  01:  // Wait for responce received
       IF ( _responseReceived )
       THEN
         // reset response received flag
        _responseReceived := FALSE;
         // update state flags
         OnUpdateStateFlags(_response.State);
         // update state flags
         OnApplyOutCmd(_response.State);
                
         // Done, Aborted or Error ?
         IF (_response.State >= CmdMessageState.DONE )
         THEN
           // Update the WorAreas in user defined system datas 
           AxesGroup.SystemData.UpdateWorAreas( Caller       := THIS^,
                                                SystemTime   := AxesGroup.State.SystemTime,
                                                WorkAreaNo   := OutCmd.WorkAreaNoReturn, 
                                                WorkAreaData := OutCmd.WorkAreaData);                     
           // set timeout
           SetTimeout(PT := _timeoutCmd, rTimer := _timerCmd);
           // inc step counter
          _stepCmd := _stepCmd + 1; 
         END_IF
       END_IF


  02: IF ( NOT Execute)
      THEN
        Reset();
      END_IF     

ELSE
  // invalid step
  SetError( ErrorID := RobotLibraryErrorIdEnum.ERR_INVALID_STEP, Overwrite := TRUE );
END_CASE


// Reset FB
IF ( NOT Execute )
THEN
  Reset(); 
END_IF
                
END_METHOD

METHOD PROTECTED OnUpdateStateFlags
VAR_INPUT
  /// Command message state
  State : CmdMessageState;
END_VAR
                  // Reset State flags
Done := FALSE;

CASE State OF

  // No operation or process is active
  CmdMessageState.EMPTY               :;
  // Created but not yet started
  CmdMessageState.CREATED             :;
  // Buffered and awaiting execution
  CmdMessageState.BUFFERED            : CommandBuffered    := TRUE;             
  // Buffered in planner for future execution
  CmdMessageState.BUFFERED_IN_PLANNER : CommandBuffered    := TRUE; 
  // Currently active and in progress
  CmdMessageState.ACTIVE              :;                                 
  // Interrupted and awaiting continuation
  CmdMessageState.INTERRUPTED         :;     
  // Requested for abort
  CmdMessageState.ABORT_REQUEST       :;
  // Successfully completed
  CmdMessageState.DONE                : Done               := TRUE;
                                        Busy               := FALSE;
  // Aborted before completion
  CmdMessageState.ABORTED             : Busy               := FALSE;
  // Encountered an error during execution
  CmdMessageState.ERROR               : Error              := TRUE;
                                        Busy               := FALSE;
END_CASE
                
END_METHOD

METHOD INTERNAL ParseResponsePayload : DINT
VAR_INPUT
  /// Response data
  ResponseData : RobotLibraryResponseDataFB;
  /// Timestamp
  Timestamp    : SystemTime;  
END_VAR
VAR
  /// Parameter count
 _parameterCnt : DINT;
END_VAR
// Table 6-200: Received CMD payload (RC to PLC) of "ReadWorkArea"
// --------------------------
// Header
// --------------------------
// Byte 00 : USINT   - ParSeq | State     
// Byte 01 : SINT    - AlarmMessageSeverity    
// Byte 02 : UINT    - AlarmMessageCode HB
// Byte 03 :         - AlarmMessageCode LB
// --------------------------
// Datablock
// --------------------------
// Byte 04 : USINT    - WorkAreaNo;
// Byte 05 : BYTE     - Reserved;
// Byte 06 : DATE     - Data.Date HW HB;
// Byte 07 :          - Data.Date HW LB;
// Byte 08 : IED_TIME - Data.Time HW HB;
// Byte 09 :          - Data.Time HW LB;
// Byte 10 :          - Data.Time LW HB;
// Byte 11 :          - Data.Time LW LB;
// Byte 12 : USINT    - Data.AreaType;
// Byte 13 : BOOL     - Data.AreaMode;
// Byte 14 : USINT    - Data.ReactionMode;
// Byte 15 : BOOL     - Data.ActiveModification;
// Byte 16 : USINT    - Data.DefinitionMode;
// Byte 17 : USINT    - Data.FrameNo;
// Byte 18 : REAL     - Data.ZeroPointX HW HB;
// Byte 19 :          - Data.ZeroPointX HW LB;
// Byte 20 :          - Data.ZeroPointX LW HB;
// Byte 21 :          - Data.ZeroPointX LW LB;
// Byte 22 : REAL     - Data.ZeroPointY HW HB;
// Byte 23 :          - Data.ZeroPointY HW LB;
// Byte 24 :          - Data.ZeroPointY LW HB;
// Byte 25 :          - Data.ZeroPointY LW LB;
// Byte 26 : REAL     - Data.ZeroPointZ HW HB;
// Byte 27 :          - Data.ZeroPointZ HW LB;
// Byte 28 :          - Data.ZeroPointZ LW HB;
// Byte 29 :          - Data.ZeroPointZ LW LB;
// Byte 30 : REAL     - Data.X1 HW HB;
// Byte 31 :          - Data.X1 HW LB;
// Byte 32 :          - Data.X1 LW HB;
// Byte 33 :          - Data.X1 LW LB;
// Byte 34 : REAL     - Data.X2 HW HB;
// Byte 35 :          - Data.X2 HW LB;
// Byte 36 :          - Data.X2 LW HB;
// Byte 37 :          - Data.X2 LW LB;
// Byte 38 : REAL     - Data.Y1 HW HB;
// Byte 39 :          - Data.Y1 HW LB;
// Byte 40 :          - Data.Y1 LW HB;
// Byte 41 :          - Data.Y1 LW LB;
// Byte 42 : REAL     - Data.Y2 HW HB;
// Byte 43 :          - Data.Y2 HW LB;
// Byte 44 :          - Data.Y2 LW HB;
// Byte 45 :          - Data.Y2 LW LB;
// Byte 46 : REAL     - Data.Z1 HW HB;
// Byte 47 :          - Data.Z1 HW LB;
// Byte 48 :          - Data.Z1 LW HB;
// Byte 49 :          - Data.Z1 LW LB;
// Byte 50 : REAL     - Data.Z2 HW HB;
// Byte 51 :          - Data.Z2 HW LB;
// Byte 52 :          - Data.Z2 LW HB;
// Byte 53 :          - Data.Z2 LW LB;
// Byte 54 : REAL     - Data.Radius HW HB;
// Byte 55 :          - Data.Radius HW LB;
// Byte 56 :          - Data.Radius LW HB;
// Byte 57 :          - Data.Radius LW LB;
// Byte 58 : REAL     - Data.JointLowerLimit.J1 HW HB;
// Byte 59 :          - Data.JointLowerLimit.J1 HW LB;
// Byte 60 :          - Data.JointLowerLimit.J1 LW HB;
// Byte 61 :          - Data.JointLowerLimit.J1 LW LB;
// Byte 62 : REAL     - Data.JointLowerLimit.J2 HW HB;
// Byte 63 :          - Data.JointLowerLimit.J2 HW LB;
// Byte 64 :          - Data.JointLowerLimit.J2 LW HB;
// Byte 65 :          - Data.JointLowerLimit.J2 LW LB;
// Byte 66 : REAL     - Data.JointLowerLimit.J3 HW HB;
// Byte 67 :          - Data.JointLowerLimit.J3 HW LB;
// Byte 68 :          - Data.JointLowerLimit.J3 LW HB;
// Byte 69 :          - Data.JointLowerLimit.J3 LW LB;
// Byte 70 : REAL     - Data.JointLowerLimit.J4 HW HB;
// Byte 71 :          - Data.JointLowerLimit.J4 HW LB;
// Byte 72 :          - Data.JointLowerLimit.J4 LW HB;
// Byte 73 :          - Data.JointLowerLimit.J4 LW LB;
// Byte 74 : REAL     - Data.JointLowerLimit.J5 HW HB;
// Byte 75 :          - Data.JointLowerLimit.J5 HW LB;
// Byte 76 :          - Data.JointLowerLimit.J5 LW HB;
// Byte 77 :          - Data.JointLowerLimit.J5 LW LB;
// Byte 78 : REAL     - Data.JointLowerLimit.J6 HW HB;
// Byte 79 :          - Data.JointLowerLimit.J6 HW LB;
// Byte 80 :          - Data.JointLowerLimit.J6 LW HB;
// Byte 81 :          - Data.JointLowerLimit.J6 LW LB;
// Byte 82 : REAL     - Data.JointLowerLimit.E1 HW HB;
// Byte 83 :          - Data.JointLowerLimit.E1 HW LB;
// Byte 84 :          - Data.JointLowerLimit.E1 LW HB;
// Byte 85 :          - Data.JointLowerLimit.E1 LW LB;
// Byte 86 : REAL     - Data.JointUpperLimit.J1 HW HB;
// Byte 87 :          - Data.JointUpperLimit.J1 HW LB;
// Byte 88 :          - Data.JointUpperLimit.J1 LW HB;
// Byte 89 :          - Data.JointUpperLimit.J1 LW LB;
// Byte 90 : REAL     - Data.JointUpperLimit.J2 HW HB;
// Byte 91 :          - Data.JointUpperLimit.J2 HW LB;
// Byte 92 :          - Data.JointUpperLimit.J2 LW HB;
// Byte 93 :          - Data.JointUpperLimit.J2 LW LB;
// Byte 94 : REAL     - Data.JointUpperLimit.J3 HW HB;
// Byte 95 :          - Data.JointUpperLimit.J3 HW LB;
// Byte 96 :          - Data.JointUpperLimit.J3 LW HB;
// Byte 97 :          - Data.JointUpperLimit.J3 LW LB;
// Byte 98 : REAL     - Data.JointUpperLimit.J4 HW HB;
// Byte 99 :          - Data.JointUpperLimit.J4 HW LB;
// Byte 100:          - Data.JointUpperLimit.J4 LW HB;
// Byte 101:          - Data.JointUpperLimit.J4 LW LB;
// Byte 102: REAL     - Data.JointUpperLimit.J5 HW HB;
// Byte 103:          - Data.JointUpperLimit.J5 HW LB;
// Byte 104:          - Data.JointUpperLimit.J5 LW HB;
// Byte 105:          - Data.JointUpperLimit.J5 LW LB;
// Byte 106: REAL     - Data.JointUpperLimit.J6 HW HB;
// Byte 107:          - Data.JointUpperLimit.J6 HW LB;
// Byte 108:          - Data.JointUpperLimit.J6 LW HB;
// Byte 109:          - Data.JointUpperLimit.J6 LW LB;
// Byte 110: REAL     - Data.JointUpperLimit.E1 HW HB;
// Byte 111:          - Data.JointUpperLimit.E1 HW LB;
// Byte 112:          - Data.JointUpperLimit.E1 LW HB;
// Byte 113:          - Data.JointUpperLimit.E1 LW LB;
// Byte 114: REAL     - Data.JointLowerLimit.E2 HW HB;
// Byte 115:          - Data.JointLowerLimit.E2 HW LB;
// Byte 116:          - Data.JointLowerLimit.E2 LW HB;
// Byte 117:          - Data.JointLowerLimit.E2 LW LB;
// Byte 118: REAL     - Data.JointLowerLimit.E3 HW HB;
// Byte 119:          - Data.JointLowerLimit.E3 HW LB;
// Byte 120:          - Data.JointLowerLimit.E3 LW HB;
// Byte 121:          - Data.JointLowerLimit.E3 LW LB;
// Byte 122: REAL     - Data.JointLowerLimit.E4 HW HB;
// Byte 123:          - Data.JointLowerLimit.E4 HW LB;
// Byte 124:          - Data.JointLowerLimit.E4 LW HB;
// Byte 125:          - Data.JointLowerLimit.E4 LW LB;
// Byte 126: REAL     - Data.JointLowerLimit.E5 HW HB;
// Byte 127:          - Data.JointLowerLimit.E5 HW LB;
// Byte 128:          - Data.JointLowerLimit.E5 LW HB;
// Byte 129:          - Data.JointLowerLimit.E5 LW LB;
// Byte 130: REAL     - Data.JointLowerLimit.E6 HW HB;
// Byte 131:          - Data.JointLowerLimit.E6 HW LB;
// Byte 132:          - Data.JointLowerLimit.E6 LW HB;
// Byte 133:          - Data.JointLowerLimit.E6 LW LB;
// Byte 134: REAL     - Data.JointUpperLimit.E2 HW HB;
// Byte 135:          - Data.JointUpperLimit.E2 HW LB;
// Byte 136:          - Data.JointUpperLimit.E2 LW HB;
// Byte 137:          - Data.JointUpperLimit.E2 LW LB;
// Byte 138: REAL     - Data.JointUpperLimit.E3 HW HB;
// Byte 139:          - Data.JointUpperLimit.E3 HW LB;
// --------------------------
                  // call base implementation to parse the header from payload buffer
ResponseData.PayloadPtr := SUPER^.ParseResponsePayload(ResponseData := ResponseData, Timestamp := Timestamp);

// copy parsed header to response
_response.ParSeq               := _rspHeader.ParSeq;
_response.State                := _rspHeader.State;
_response.AlarmMessageSeverity := _rspHeader.AlarmMessageSeverity;
_response.AlarmMessageCode     := _rspHeader.AlarmMessageCode;


// Check payload remaining ? 
IF ( ResponseData.IsPayloadRemaining)
THEN  
  // Get Response.WorkAreaNoReturn
 _response.WorkAreaNoReturn := ResponseData.GetUsint();
  // inc parameter counter
 _parameterCnt := _parameterCnt + 1;
END_IF


// Check payload remaining ? 
IF ( ResponseData.IsPayloadRemaining)
THEN  
  // Get Response.Reserve
 _response.Reserve := ResponseData.GetByte();
  // inc parameter counter
 _parameterCnt := _parameterCnt + 1;
END_IF


// Check payload remaining ? 
IF ( ResponseData.IsPayloadRemaining)
THEN  
  // Get Response.WorkAreaData.Timestamp.IEC_DATE
 _response.WorkAreaData.Timestamp.IEC_DATE := ResponseData.GetIecDate();
  // inc parameter counter
 _parameterCnt := _parameterCnt + 1;
END_IF


// Check payload remaining ? 
IF ( ResponseData.IsPayloadRemaining)
THEN  
  // Get Response.WorkAreaData.Timestamp.IEC_TIME
 _response.WorkAreaData.Timestamp.IEC_TIME := ResponseData.GetIecTime();
  // inc parameter counter
 _parameterCnt := _parameterCnt + 1;
END_IF


// Check payload remaining ? 
IF ( ResponseData.IsPayloadRemaining)
THEN  
  // Get Response.WorkAreaData.AreaType
 _response.WorkAreaData.AreaType := ResponseData.GetUsint();
  // inc parameter counter
 _parameterCnt := _parameterCnt + 1;
END_IF


// Check payload remaining ? 
IF ( ResponseData.IsPayloadRemaining)
THEN  
  // Get Response.WorkAreaData.AreaMode
 _response.WorkAreaData.AreaMode := ResponseData.GetBool();
  // inc parameter counter
 _parameterCnt := _parameterCnt + 1;
END_IF


// Check payload remaining ? 
IF ( ResponseData.IsPayloadRemaining)
THEN  
  // Get Response.WorkAreaData.ReactionMode
 _response.WorkAreaData.ReactionMode := ResponseData.GetUsint();
  // inc parameter counter
 _parameterCnt := _parameterCnt + 1;
END_IF


// Check payload remaining ? 
IF ( ResponseData.IsPayloadRemaining)
THEN  
  // Get Response.WorkAreaData.ActiveModification
 _response.WorkAreaData.ActiveModification := ResponseData.GetBool();
  // inc parameter counter
 _parameterCnt := _parameterCnt + 1;
END_IF


// Check payload remaining ? 
IF ( ResponseData.IsPayloadRemaining)
THEN  
  // Get Response.WorkAreaData.DefinitionMode
 _response.WorkAreaData.DefinitionMode := ResponseData.GetUsint();
  // inc parameter counter
 _parameterCnt := _parameterCnt + 1;
END_IF


// Check payload remaining ? 
IF ( ResponseData.IsPayloadRemaining)
THEN  
  // Get Response.WorkAreaData.FrameNo
 _response.WorkAreaData.FrameNo := ResponseData.GetUsint();
  // inc parameter counter
 _parameterCnt := _parameterCnt + 1;
END_IF


// Check payload remaining ? 
IF ( ResponseData.IsPayloadRemaining)
THEN  
  // Get Response.WorkAreaData.ZeroPointX
 _response.WorkAreaData.ZeroPointX := ResponseData.GetReal();
  // inc parameter counter
 _parameterCnt := _parameterCnt + 1;
END_IF


// Check payload remaining ? 
IF ( ResponseData.IsPayloadRemaining)
THEN  
  // Get Response.WorkAreaData.ZeroPointY
 _response.WorkAreaData.ZeroPointY := ResponseData.GetReal();
  // inc parameter counter
 _parameterCnt := _parameterCnt + 1;
END_IF


// Check payload remaining ? 
IF ( ResponseData.IsPayloadRemaining)
THEN  
  // Get Response.WorkAreaData.ZeroPointZ
 _response.WorkAreaData.ZeroPointZ := ResponseData.GetReal();
  // inc parameter counter
 _parameterCnt := _parameterCnt + 1;
END_IF


// Check payload remaining ? 
IF ( ResponseData.IsPayloadRemaining)
THEN  
  // Get Response.WorkAreaData.X.LowerLimit
 _response.WorkAreaData.X.LowerLimit := ResponseData.GetReal();
  // inc parameter counter
 _parameterCnt := _parameterCnt + 1;
END_IF


// Check payload remaining ? 
IF ( ResponseData.IsPayloadRemaining)
THEN  
  // Get Response.WorkAreaData.X.UpperLimit
 _response.WorkAreaData.X.UpperLimit := ResponseData.GetReal();
  // inc parameter counter
 _parameterCnt := _parameterCnt + 1;
END_IF


// Check payload remaining ? 
IF ( ResponseData.IsPayloadRemaining)
THEN  
  // Get Response.WorkAreaData.Y.LowerLimit
 _response.WorkAreaData.Y.LowerLimit := ResponseData.GetReal();
  // inc parameter counter
 _parameterCnt := _parameterCnt + 1;
END_IF


// Check payload remaining ? 
IF ( ResponseData.IsPayloadRemaining)
THEN  
  // Get Response.WorkAreaData.Y.UpperLimit
 _response.WorkAreaData.Y.UpperLimit := ResponseData.GetReal();
  // inc parameter counter
 _parameterCnt := _parameterCnt + 1;
END_IF


// Check payload remaining ? 
IF ( ResponseData.IsPayloadRemaining)
THEN  
  // Get Response.WorkAreaData.Z.LowerLimit
 _response.WorkAreaData.Z.LowerLimit := ResponseData.GetReal();
  // inc parameter counter
 _parameterCnt := _parameterCnt + 1;
END_IF


// Check payload remaining ? 
IF ( ResponseData.IsPayloadRemaining)
THEN  
  // Get Response.WorkAreaData.Z.UpperLimit
 _response.WorkAreaData.Z.UpperLimit := ResponseData.GetReal();
  // inc parameter counter
 _parameterCnt := _parameterCnt + 1;
END_IF


// Check payload remaining ? 
IF ( ResponseData.IsPayloadRemaining)
THEN  
  // Get Response.WorkAreaData.Radiust
 _response.WorkAreaData.Radius := ResponseData.GetReal();
  // inc parameter counter
 _parameterCnt := _parameterCnt + 1;
END_IF


// Check payload remaining ? 
IF ( ResponseData.IsPayloadRemaining)
THEN  
  // Get Response.WorkAreaData.J1Limit.LowerLimit
 _response.WorkAreaData.J1Limit.LowerLimit := ResponseData.GetReal();
  // inc parameter counter
 _parameterCnt := _parameterCnt + 1;
END_IF


// Check payload remaining ? 
IF ( ResponseData.IsPayloadRemaining)
THEN  
  // Get Response.WorkAreaData.J2Limit.LowerLimit
 _response.WorkAreaData.J2Limit.LowerLimit := ResponseData.GetReal();
  // inc parameter counter
 _parameterCnt := _parameterCnt + 1;
END_IF


// Check payload remaining ? 
IF ( ResponseData.IsPayloadRemaining)
THEN  
  // Get Response.WorkAreaData.J3Limit.LowerLimit
 _response.WorkAreaData.J3Limit.LowerLimit := ResponseData.GetReal();
  // inc parameter counter
 _parameterCnt := _parameterCnt + 1;
END_IF


// Check payload remaining ? 
IF ( ResponseData.IsPayloadRemaining)
THEN  
  // Get Response.WorkAreaData.J4Limit.LowerLimit
 _response.WorkAreaData.J4Limit.LowerLimit := ResponseData.GetReal();
  // inc parameter counter
 _parameterCnt := _parameterCnt + 1;
END_IF


// Check payload remaining ? 
IF ( ResponseData.IsPayloadRemaining)
THEN  
  // Get Response.WorkAreaData.J5Limit.LowerLimit
 _response.WorkAreaData.J5Limit.LowerLimit := ResponseData.GetReal();
  // inc parameter counter
 _parameterCnt := _parameterCnt + 1;
END_IF


// Check payload remaining ? 
IF ( ResponseData.IsPayloadRemaining)
THEN  
  // Get Response.WorkAreaData.J6Limit.LowerLimit
 _response.WorkAreaData.J6Limit.LowerLimit := ResponseData.GetReal();
  // inc parameter counter
 _parameterCnt := _parameterCnt + 1;
END_IF


// Check payload remaining ? 
IF ( ResponseData.IsPayloadRemaining)
THEN  
  // Get Response.WorkAreaData.E1Limit.LowerLimit
 _response.WorkAreaData.E1Limit.LowerLimit := ResponseData.GetReal();
  // inc parameter counter
 _parameterCnt := _parameterCnt + 1;
END_IF


// Check payload remaining ? 
IF ( ResponseData.IsPayloadRemaining)
THEN  
  // Get Response.WorkAreaData.J1Limit.UpperLimit
 _response.WorkAreaData.J1Limit.UpperLimit := ResponseData.GetReal();
  // inc parameter counter
 _parameterCnt := _parameterCnt + 1;
END_IF


// Check payload remaining ? 
IF ( ResponseData.IsPayloadRemaining)
THEN  
  // Get Response.WorkAreaData.J2Limit.UpperLimit
 _response.WorkAreaData.J2Limit.UpperLimit := ResponseData.GetReal();
  // inc parameter counter
 _parameterCnt := _parameterCnt + 1;
END_IF


// Check payload remaining ? 
IF ( ResponseData.IsPayloadRemaining)
THEN  
  // Get Response.WorkAreaData.J3Limit.UpperLimit
 _response.WorkAreaData.J3Limit.UpperLimit := ResponseData.GetReal();
  // inc parameter counter
 _parameterCnt := _parameterCnt + 1;
END_IF


// Check payload remaining ? 
IF ( ResponseData.IsPayloadRemaining)
THEN  
  // Get Response.WorkAreaData.J4Limit.UpperLimit
 _response.WorkAreaData.J4Limit.UpperLimit := ResponseData.GetReal();
  // inc parameter counter
 _parameterCnt := _parameterCnt + 1;
END_IF


// Check payload remaining ? 
IF ( ResponseData.IsPayloadRemaining)
THEN  
  // Get Response.WorkAreaData.J5Limit.UpperLimit
 _response.WorkAreaData.J5Limit.UpperLimit := ResponseData.GetReal();
  // inc parameter counter
 _parameterCnt := _parameterCnt + 1;
END_IF


// Check payload remaining ? 
IF ( ResponseData.IsPayloadRemaining)
THEN  
  // Get Response.WorkAreaData.J6Limit.UpperLimit
 _response.WorkAreaData.J6Limit.UpperLimit := ResponseData.GetReal();
  // inc parameter counter
 _parameterCnt := _parameterCnt + 1;
END_IF


// Check payload remaining ? 
IF ( ResponseData.IsPayloadRemaining)
THEN  
  // Get Response.WorkAreaData.E1Limit.UpperLimit
 _response.WorkAreaData.E1Limit.UpperLimit := ResponseData.GetReal();
  // inc parameter counter
 _parameterCnt := _parameterCnt + 1;
END_IF


// Check payload remaining ? 
IF ( ResponseData.IsPayloadRemaining)
THEN  
  // Get Response.WorkAreaData.E2Limit.LowerLimit
 _response.WorkAreaData.E2Limit.LowerLimit := ResponseData.GetReal();
  // inc parameter counter
 _parameterCnt := _parameterCnt + 1;
END_IF


// Check payload remaining ? 
IF ( ResponseData.IsPayloadRemaining)
THEN  
  // Get Response.WorkAreaData.E3Limit.LowerLimit
 _response.WorkAreaData.E3Limit.LowerLimit := ResponseData.GetReal();
  // inc parameter counter
 _parameterCnt := _parameterCnt + 1;
END_IF


// Check payload remaining ? 
IF ( ResponseData.IsPayloadRemaining)
THEN  
  // Get Response.WorkAreaData.E4Limit.LowerLimit
 _response.WorkAreaData.E4Limit.LowerLimit := ResponseData.GetReal();
  // inc parameter counter
 _parameterCnt := _parameterCnt + 1;
END_IF


// Check payload remaining ? 
IF ( ResponseData.IsPayloadRemaining)
THEN  
  // Get Response.WorkAreaData.E5Limit.LowerLimit
 _response.WorkAreaData.E5Limit.LowerLimit := ResponseData.GetReal();
  // inc parameter counter
 _parameterCnt := _parameterCnt + 1;
END_IF


// Check payload remaining ? 
IF ( ResponseData.IsPayloadRemaining)
THEN  
  // Get Response.WorkAreaData.E6Limit.LowerLimit
 _response.WorkAreaData.E6Limit.LowerLimit := ResponseData.GetReal();
  // inc parameter counter
 _parameterCnt := _parameterCnt + 1;
END_IF


// Check payload remaining ? 
IF ( ResponseData.IsPayloadRemaining)
THEN  
  // Get Response.WorkAreaData.E2Limit.UpperLimit
 _response.WorkAreaData.E2Limit.UpperLimit := ResponseData.GetReal();
  // inc parameter counter
 _parameterCnt := _parameterCnt + 1;
END_IF


// Check payload remaining ? 
IF ( ResponseData.IsPayloadRemaining)
THEN  
  // Get Response.WorkAreaData.E3Limit.UpperLimit
 _response.WorkAreaData.E3Limit.UpperLimit := ResponseData.GetReal();
  // inc parameter counter
 _parameterCnt := _parameterCnt + 1;
END_IF


// Check payload remaining ? 
IF ( ResponseData.IsPayloadRemaining)
THEN  
  // Get Response.WorkAreaData.E4Limit.UpperLimit
 _response.WorkAreaData.E4Limit.UpperLimit := ResponseData.GetReal();
  // inc parameter counter
 _parameterCnt := _parameterCnt + 1;
END_IF


// Check payload remaining ? 
IF ( ResponseData.IsPayloadRemaining)
THEN  
  // Get Response.WorkAreaData.E5Limit.UpperLimit
 _response.WorkAreaData.E5Limit.UpperLimit := ResponseData.GetReal();
  // inc parameter counter
 _parameterCnt := _parameterCnt + 1;
END_IF


// Check payload remaining ? 
IF ( ResponseData.IsPayloadRemaining)
THEN  
  // Get Response.WorkAreaData.E6Limit.UpperLimit
 _response.WorkAreaData.E6Limit.UpperLimit := ResponseData.GetReal();
  // inc parameter counter
 _parameterCnt := _parameterCnt + 1;
END_IF


// Check payload remaining ? 
IF ( ResponseData.IsPayloadRemaining)
THEN  
  // Get Response.DataChanged
 _response.DataChanged := ResponseData.GetBool();
  // inc parameter counter
 _parameterCnt := _parameterCnt + 1;
END_IF



// Create logging
ParseResponsePayloadLog(ResponseData := ResponseData, Timestamp := Timestamp, ParameterCnt := _parameterCnt);
                
END_METHOD

METHOD INTERNAL ParseResponsePayloadLog
VAR_INPUT
  /// Response data
  ResponseData : RobotLibraryResponseDataFB;
  /// Timestamp
  Timestamp    : SystemTime;  
  /// Parameter count
  ParameterCnt : DINT;
END_VAR
                  // Create log entry for Parameter start
CreateLogMessagePara1 ( Timestamp   := Timestamp,
                        MessageType := MessageType.CMD,
                        Severity    := Severity.DEBUG,
                        MessageCode := 0,
                        MessageText := '{1} parameter(s) to parse from the response data:',
                        Para1       := DINT_TO_STRING(ParameterCnt));
                        

// Return if no parameter is remaining...
IF ( ParameterCnt = 0 ) THEN RETURN; END_IF
// dec remaining parameter(s)                        
ParameterCnt := ParameterCnt - 1;
// Create log entry for WorkAreaNoReturn
CreateLogMessagePara1 ( Timestamp   := Timestamp,
                        MessageType := MessageType.CMD,
                        Severity    := Severity.DEBUG,
                        MessageCode := 0,
                        MessageText := 'Response.WorkAreaNoReturn = {1}',
                        Para1       :=  USINT_TO_STRING(_response.WorkAreaNoReturn));


// Return if no parameter is remaining...
IF ( ParameterCnt = 0 ) THEN RETURN; END_IF
// dec remaining parameter(s)                        
ParameterCnt := ParameterCnt - 1;
// Create log entry for Reserve
CreateLogMessagePara1 ( Timestamp   := Timestamp,
                        MessageType := MessageType.CMD,
                        Severity    := Severity.DEBUG,
                        MessageCode := 0,
                        MessageText := 'Response.Reserve = {1}',
                        Para1       :=  BYTE_TO_STRING(_response.Reserve));


// Return if no parameter is remaining...
IF ( ParameterCnt = 0 ) THEN RETURN; END_IF
// dec remaining parameter(s)                        
ParameterCnt := ParameterCnt - 1;
// Create log entry for WorkAreaData.Timestamp.IEC_DATE
CreateLogMessagePara1 ( Timestamp   := Timestamp,
                        MessageType := MessageType.CMD,
                        Severity    := Severity.DEBUG,
                        MessageCode := 0,
                        MessageText := 'Response.WorkAreaData.Timestamp.IEC_DATE = {1}',
                        Para1       :=  IEC_DATE_TO_STRING(_response.WorkAreaData.Timestamp.IEC_DATE));


// Return if no parameter is remaining...
IF ( ParameterCnt = 0 ) THEN RETURN; END_IF
// dec remaining parameter(s)                        
ParameterCnt := ParameterCnt - 1;
// Create log entry for WorkAreaData.Timestamp.IEC_TIME
CreateLogMessagePara1 ( Timestamp   := Timestamp,
                        MessageType := MessageType.CMD,
                        Severity    := Severity.DEBUG,
                        MessageCode := 0,
                        MessageText := 'Response.WorkAreaData.Timestamp.IEC_TIME = {1}',
                        Para1       :=  IEC_TIME_TO_STRING(_response.WorkAreaData.Timestamp.IEC_TIME));


// Return if no parameter is remaining...
IF ( ParameterCnt = 0 ) THEN RETURN; END_IF
// dec remaining parameter(s)                        
ParameterCnt := ParameterCnt - 1;
// Create log entry for WorkAreaData.AreaType
CreateLogMessagePara1 ( Timestamp   := Timestamp,
                        MessageType := MessageType.CMD,
                        Severity    := Severity.DEBUG,
                        MessageCode := 0,
                        MessageText := 'Response.WorkAreaData.AreaType = {1}',
                        Para1       :=  USINT_TO_STRING(_response.WorkAreaData.AreaType));


// Return if no parameter is remaining...
IF ( ParameterCnt = 0 ) THEN RETURN; END_IF
// dec remaining parameter(s)                        
ParameterCnt := ParameterCnt - 1;
// Create log entry for WorkAreaData.AreaMode
CreateLogMessagePara1 ( Timestamp   := Timestamp,
                        MessageType := MessageType.CMD,
                        Severity    := Severity.DEBUG,
                        MessageCode := 0,
                        MessageText := 'Response.WorkAreaData.AreaMode = {1}',
                        Para1       :=  BOOL_TO_STRING(_response.WorkAreaData.AreaMode));
                        

// Return if no parameter is remaining...
IF ( ParameterCnt = 0 ) THEN RETURN; END_IF
// dec remaining parameter(s)                        
ParameterCnt := ParameterCnt - 1;
// Create log entry for WorkAreaData.ReactionMode
CreateLogMessagePara1 ( Timestamp   := Timestamp,
                        MessageType := MessageType.CMD,
                        Severity    := Severity.DEBUG,
                        MessageCode := 0,
                        MessageText := 'Response.WorkAreaData.ReactionMode = {1}',
                        Para1       :=  WORK_AREA_REACTION_MODE_TO_STRING(_response.WorkAreaData.ReactionMode));


// Return if no parameter is remaining...
IF ( ParameterCnt = 0 ) THEN RETURN; END_IF
// dec remaining parameter(s)                        
ParameterCnt := ParameterCnt - 1;
// Create log entry for WorkAreaData.ActiveModification
CreateLogMessagePara1 ( Timestamp   := Timestamp,
                        MessageType := MessageType.CMD,
                        Severity    := Severity.DEBUG,
                        MessageCode := 0,
                        MessageText := 'Response.WorkAreaData.ActiveModification = {1}',
                        Para1       :=  BOOL_TO_STRING(_response.WorkAreaData.ActiveModification));


// Return if no parameter is remaining...
IF ( ParameterCnt = 0 ) THEN RETURN; END_IF
// dec remaining parameter(s)                        
ParameterCnt := ParameterCnt - 1;
// Create log entry for WorkAreaData.DefinitionMode
CreateLogMessagePara1 ( Timestamp   := Timestamp,
                        MessageType := MessageType.CMD,
                        Severity    := Severity.DEBUG,
                        MessageCode := 0,
                        MessageText := 'Response.WorkAreaData.DefinitionMode = {1}',
                        Para1       := DEFINITION_MODE_TO_STRING(_response.WorkAreaData.DefinitionMode));


// Return if no parameter is remaining...
IF ( ParameterCnt = 0 ) THEN RETURN; END_IF
// dec remaining parameter(s)                        
ParameterCnt := ParameterCnt - 1;
// Create log entry for WorkAreaData.FrameNo
CreateLogMessagePara1 ( Timestamp   := Timestamp,
                        MessageType := MessageType.CMD,
                        Severity    := Severity.DEBUG,
                        MessageCode := 0,
                        MessageText := 'Response.WorkAreaData.FrameNo = {1}',
                        Para1       :=  USINT_TO_STRING(_response.WorkAreaData.FrameNo));


// Return if no parameter is remaining...
IF ( ParameterCnt = 0 ) THEN RETURN; END_IF
// dec remaining parameter(s)                        
ParameterCnt := ParameterCnt - 1;
// Create log entry for WorkAreaData.ZeroPointX
CreateLogMessagePara1 ( Timestamp   := Timestamp,
                        MessageType := MessageType.CMD,
                        Severity    := Severity.DEBUG,
                        MessageCode := 0,
                        MessageText := 'Response.WorkAreaData.ZeroPointX = {1}',
                        Para1       :=  REAL_TO_STRING(_response.WorkAreaData.ZeroPointX));


// Return if no parameter is remaining...
IF ( ParameterCnt = 0 ) THEN RETURN; END_IF
// dec remaining parameter(s)                        
ParameterCnt := ParameterCnt - 1;
// Create log entry for WorkAreaData.ZeroPointY
CreateLogMessagePara1 ( Timestamp   := Timestamp,
                        MessageType := MessageType.CMD,
                        Severity    := Severity.DEBUG,
                        MessageCode := 0,
                        MessageText := 'Response.WorkAreaData.ZeroPointY = {1}',
                        Para1       :=  REAL_TO_STRING(_response.WorkAreaData.ZeroPointY));


// Return if no parameter is remaining...
IF ( ParameterCnt = 0 ) THEN RETURN; END_IF
// dec remaining parameter(s)                        
ParameterCnt := ParameterCnt - 1;
// Create log entry for WorkAreaData.ZeroPointZ
CreateLogMessagePara1 ( Timestamp   := Timestamp,
                        MessageType := MessageType.CMD,
                        Severity    := Severity.DEBUG,
                        MessageCode := 0,
                        MessageText := 'Response.WorkAreaData.ZeroPointZ = {1}',
                        Para1       :=  REAL_TO_STRING(_response.WorkAreaData.ZeroPointZ));


// Return if no parameter is remaining...
IF ( ParameterCnt = 0 ) THEN RETURN; END_IF
// dec remaining parameter(s)                        
ParameterCnt := ParameterCnt - 1;
// Create log entry for WorkAreaData.X.LowerLimit
CreateLogMessagePara1 ( Timestamp   := Timestamp,
                        MessageType := MessageType.CMD,
                        Severity    := Severity.DEBUG,
                        MessageCode := 0,
                        MessageText := 'Response.WorkAreaData.X.LowerLimit = {1}',
                        Para1       :=  REAL_TO_STRING(_response.WorkAreaData.X.LowerLimit));


// Return if no parameter is remaining...
IF ( ParameterCnt = 0 ) THEN RETURN; END_IF
// dec remaining parameter(s)                        
ParameterCnt := ParameterCnt - 1;
// Create log entry for WorkAreaData.X.UpperLimit
CreateLogMessagePara1 ( Timestamp   := Timestamp,
                        MessageType := MessageType.CMD,
                        Severity    := Severity.DEBUG,
                        MessageCode := 0,
                        MessageText := 'Response.WorkAreaData.X.UpperLimit = {1}',
                        Para1       :=  REAL_TO_STRING(_response.WorkAreaData.X.UpperLimit));


// Return if no parameter is remaining...
IF ( ParameterCnt = 0 ) THEN RETURN; END_IF
// dec remaining parameter(s)                        
ParameterCnt := ParameterCnt - 1;
// Create log entry for WorkAreaData.Y.LowerLimit
CreateLogMessagePara1 ( Timestamp   := Timestamp,
                        MessageType := MessageType.CMD,
                        Severity    := Severity.DEBUG,
                        MessageCode := 0,
                        MessageText := 'Response.WorkAreaData.Y.LowerLimit = {1}',
                        Para1       :=  REAL_TO_STRING(_response.WorkAreaData.Y.LowerLimit));


// Return if no parameter is remaining...
IF ( ParameterCnt = 0 ) THEN RETURN; END_IF
// dec remaining parameter(s)                        
ParameterCnt := ParameterCnt - 1;
// Create log entry for WorkAreaData.Y.UpperLimit
CreateLogMessagePara1 ( Timestamp   := Timestamp,
                        MessageType := MessageType.CMD,
                        Severity    := Severity.DEBUG,
                        MessageCode := 0,
                        MessageText := 'Response.WorkAreaData.Y.UpperLimit = {1}',
                        Para1       :=  REAL_TO_STRING(_response.WorkAreaData.Y.UpperLimit));


// Return if no parameter is remaining...
IF ( ParameterCnt = 0 ) THEN RETURN; END_IF
// dec remaining parameter(s)                        
ParameterCnt := ParameterCnt - 1;
// Create log entry for WorkAreaData.Z.LowerLimit
CreateLogMessagePara1 ( Timestamp   := Timestamp,
                        MessageType := MessageType.CMD,
                        Severity    := Severity.DEBUG,
                        MessageCode := 0,
                        MessageText := 'Response.WorkAreaData.Z.LowerLimit = {1}',
                        Para1       :=  REAL_TO_STRING(_response.WorkAreaData.Z.LowerLimit));


// Return if no parameter is remaining...
IF ( ParameterCnt = 0 ) THEN RETURN; END_IF
// dec remaining parameter(s)                        
ParameterCnt := ParameterCnt - 1;
// Create log entry for WorkAreaData.Z.UpperLimit
CreateLogMessagePara1 ( Timestamp   := Timestamp,
                        MessageType := MessageType.CMD,
                        Severity    := Severity.DEBUG,
                        MessageCode := 0,
                        MessageText := 'Response.WorkAreaData.Z.UpperLimit = {1}',
                        Para1       :=  REAL_TO_STRING(_response.WorkAreaData.Z.UpperLimit));


// Return if no parameter is remaining...
IF ( ParameterCnt = 0 ) THEN RETURN; END_IF
// dec remaining parameter(s)                        
ParameterCnt := ParameterCnt - 1;
// Create log entry for WorkAreaData.Radius
CreateLogMessagePara1 ( Timestamp   := Timestamp,
                        MessageType := MessageType.CMD,
                        Severity    := Severity.DEBUG,
                        MessageCode := 0,
                        MessageText := 'Response.WorkAreaData.Radius = {1}',
                        Para1       :=  REAL_TO_STRING(_response.WorkAreaData.Radius));


// Return if no parameter is remaining...
IF ( ParameterCnt = 0 ) THEN RETURN; END_IF
// dec remaining parameter(s)                        
ParameterCnt := ParameterCnt - 1;
// Create log entry for WorkAreaData.J1Limit.LowerLimit
CreateLogMessagePara1 ( Timestamp   := Timestamp,
                        MessageType := MessageType.CMD,
                        Severity    := Severity.DEBUG,
                        MessageCode := 0,
                        MessageText := 'Response.WorkAreaData.J1Limit.LowerLimit = {1}',
                        Para1       :=  REAL_TO_STRING(_response.WorkAreaData.J1Limit.LowerLimit));


// Return if no parameter is remaining...
IF ( ParameterCnt = 0 ) THEN RETURN; END_IF
// dec remaining parameter(s)                        
ParameterCnt := ParameterCnt - 1;
// Create log entry for WorkAreaData.J2Limit.LowerLimit
CreateLogMessagePara1 ( Timestamp   := Timestamp,
                        MessageType := MessageType.CMD,
                        Severity    := Severity.DEBUG,
                        MessageCode := 0,
                        MessageText := 'Response.WorkAreaData.J2Limit.LowerLimit = {1}',
                        Para1       :=  REAL_TO_STRING(_response.WorkAreaData.J2Limit.LowerLimit));


// Return if no parameter is remaining...
IF ( ParameterCnt = 0 ) THEN RETURN; END_IF
// dec remaining parameter(s)                        
ParameterCnt := ParameterCnt - 1;
// Create log entry for WorkAreaData.J3Limit.LowerLimit
CreateLogMessagePara1 ( Timestamp   := Timestamp,
                        MessageType := MessageType.CMD,
                        Severity    := Severity.DEBUG,
                        MessageCode := 0,
                        MessageText := 'Response.WorkAreaData.J3Limit.LowerLimit = {1}',
                        Para1       :=  REAL_TO_STRING(_response.WorkAreaData.J3Limit.LowerLimit));

// Return if no parameter is remaining...
IF ( ParameterCnt = 0 ) THEN RETURN; END_IF
// dec remaining parameter(s)                        
ParameterCnt := ParameterCnt - 1;
// Create log entry for WorkAreaData.J4Limit.LowerLimit
CreateLogMessagePara1 ( Timestamp   := Timestamp,
                        MessageType := MessageType.CMD,
                        Severity    := Severity.DEBUG,
                        MessageCode := 0,
                        MessageText := 'Response.WorkAreaData.J4Limit.LowerLimit = {1}',
                        Para1       :=  REAL_TO_STRING(_response.WorkAreaData.J4Limit.LowerLimit));


// Return if no parameter is remaining...
IF ( ParameterCnt = 0 ) THEN RETURN; END_IF
// dec remaining parameter(s)                        
ParameterCnt := ParameterCnt - 1;
// Create log entry for WorkAreaData.J5Limit.LowerLimit
CreateLogMessagePara1 ( Timestamp   := Timestamp,
                        MessageType := MessageType.CMD,
                        Severity    := Severity.DEBUG,
                        MessageCode := 0,
                        MessageText := 'Response.WorkAreaData.J5Limit.LowerLimit = {1}',
                        Para1       :=  REAL_TO_STRING(_response.WorkAreaData.J5Limit.LowerLimit));


// Return if no parameter is remaining...
IF ( ParameterCnt = 0 ) THEN RETURN; END_IF
// dec remaining parameter(s)                        
ParameterCnt := ParameterCnt - 1;
// Create log entry for WorkAreaData.J6Limit.LowerLimit
CreateLogMessagePara1 ( Timestamp   := Timestamp,
                        MessageType := MessageType.CMD,
                        Severity    := Severity.DEBUG,
                        MessageCode := 0,
                        MessageText := 'Response.WorkAreaData.J6Limit.LowerLimit = {1}',
                        Para1       :=  REAL_TO_STRING(_response.WorkAreaData.J6Limit.LowerLimit));


// Return if no parameter is remaining...
IF ( ParameterCnt = 0 ) THEN RETURN; END_IF
// dec remaining parameter(s)                        
ParameterCnt := ParameterCnt - 1;
// Create log entry for WorkAreaData.E1Limit.LowerLimit
CreateLogMessagePara1 ( Timestamp   := Timestamp,
                        MessageType := MessageType.CMD,
                        Severity    := Severity.DEBUG,
                        MessageCode := 0,
                        MessageText := 'Response.WorkAreaData.E1Limit.LowerLimit = {1}',
                        Para1       :=  REAL_TO_STRING(_response.WorkAreaData.E1Limit.LowerLimit));


// Return if no parameter is remaining...
IF ( ParameterCnt = 0 ) THEN RETURN; END_IF
// dec remaining parameter(s)                        
ParameterCnt := ParameterCnt - 1;
// Create log entry for WorkAreaData.J1Limit.UpperLimit
CreateLogMessagePara1 ( Timestamp   := Timestamp,
                        MessageType := MessageType.CMD,
                        Severity    := Severity.DEBUG,
                        MessageCode := 0,
                        MessageText := 'Response.WorkAreaData.J1Limit.UpperLimit = {1}',
                        Para1       :=  REAL_TO_STRING(_response.WorkAreaData.J1Limit.UpperLimit));


// Return if no parameter is remaining...
IF ( ParameterCnt = 0 ) THEN RETURN; END_IF
// dec remaining parameter(s)                        
ParameterCnt := ParameterCnt - 1;
// Create log entry for WorkAreaData.J2Limit.UpperLimit
CreateLogMessagePara1 ( Timestamp   := Timestamp,
                        MessageType := MessageType.CMD,
                        Severity    := Severity.DEBUG,
                        MessageCode := 0,
                        MessageText := 'Response.WorkAreaData.J2Limit.UpperLimit = {1}',
                        Para1       :=  REAL_TO_STRING(_response.WorkAreaData.J2Limit.UpperLimit));


// Return if no parameter is remaining...
IF ( ParameterCnt = 0 ) THEN RETURN; END_IF
// dec remaining parameter(s)                        
ParameterCnt := ParameterCnt - 1;
// Create log entry for WorkAreaData.J3Limit.UpperLimit
CreateLogMessagePara1 ( Timestamp   := Timestamp,
                        MessageType := MessageType.CMD,
                        Severity    := Severity.DEBUG,
                        MessageCode := 0,
                        MessageText := 'Response.WorkAreaData.J3Limit.UpperLimit = {1}',
                        Para1       :=  REAL_TO_STRING(_response.WorkAreaData.J3Limit.UpperLimit));


// Return if no parameter is remaining...
IF ( ParameterCnt = 0 ) THEN RETURN; END_IF
// dec remaining parameter(s)                        
ParameterCnt := ParameterCnt - 1;
// Create log entry for WorkAreaData.J4Limit.UpperLimit
CreateLogMessagePara1 ( Timestamp   := Timestamp,
                        MessageType := MessageType.CMD,
                        Severity    := Severity.DEBUG,
                        MessageCode := 0,
                        MessageText := 'Response.WorkAreaData.J4Limit.UpperLimit = {1}',
                        Para1       :=  REAL_TO_STRING(_response.WorkAreaData.J4Limit.UpperLimit));


// Return if no parameter is remaining...
IF ( ParameterCnt = 0 ) THEN RETURN; END_IF
// dec remaining parameter(s)                        
ParameterCnt := ParameterCnt - 1;
// Create log entry for WorkAreaData.J5Limit.UpperLimit
CreateLogMessagePara1 ( Timestamp   := Timestamp,
                        MessageType := MessageType.CMD,
                        Severity    := Severity.DEBUG,
                        MessageCode := 0,
                        MessageText := 'Response.WorkAreaData.J5Limit.UpperLimit = {1}',
                        Para1       :=  REAL_TO_STRING(_response.WorkAreaData.J5Limit.UpperLimit));


// Return if no parameter is remaining...
IF ( ParameterCnt = 0 ) THEN RETURN; END_IF
// dec remaining parameter(s)                        
ParameterCnt := ParameterCnt - 1;
// Create log entry for WorkAreaData.J6Limit.UpperLimit
CreateLogMessagePara1 ( Timestamp   := Timestamp,
                        MessageType := MessageType.CMD,
                        Severity    := Severity.DEBUG,
                        MessageCode := 0,
                        MessageText := 'Response.WorkAreaData.J6Limit.UpperLimit = {1}',
                        Para1       :=  REAL_TO_STRING(_response.WorkAreaData.J6Limit.UpperLimit));


// Return if no parameter is remaining...
IF ( ParameterCnt = 0 ) THEN RETURN; END_IF
// dec remaining parameter(s)                        
ParameterCnt := ParameterCnt - 1;
// Create log entry for WorkAreaData.E1Limit.UpperLimit
CreateLogMessagePara1 ( Timestamp   := Timestamp,
                        MessageType := MessageType.CMD,
                        Severity    := Severity.DEBUG,
                        MessageCode := 0,
                        MessageText := 'Response.WorkAreaData.E1Limit.UpperLimit = {1}',
                        Para1       :=  REAL_TO_STRING(_response.WorkAreaData.E1Limit.UpperLimit));


// Return if no parameter is remaining...
IF ( ParameterCnt = 0 ) THEN RETURN; END_IF
// dec remaining parameter(s)                        
ParameterCnt := ParameterCnt - 1;
// Create log entry for WorkAreaData.E2Limit.LowerLimit
CreateLogMessagePara1 ( Timestamp   := Timestamp,
                        MessageType := MessageType.CMD,
                        Severity    := Severity.DEBUG,
                        MessageCode := 0,
                        MessageText := 'Response.WorkAreaData.E2Limit.LowerLimit = {1}',
                        Para1       :=  REAL_TO_STRING(_response.WorkAreaData.E2Limit.LowerLimit));


// Return if no parameter is remaining...
IF ( ParameterCnt = 0 ) THEN RETURN; END_IF
// dec remaining parameter(s)                        
ParameterCnt := ParameterCnt - 1;
// Create log entry for WorkAreaData.E3Limit.LowerLimit
CreateLogMessagePara1 ( Timestamp   := Timestamp,
                        MessageType := MessageType.CMD,
                        Severity    := Severity.DEBUG,
                        MessageCode := 0,
                        MessageText := 'Response.WorkAreaData.E3Limit.LowerLimit = {1}',
                        Para1       :=  REAL_TO_STRING(_response.WorkAreaData.E3Limit.LowerLimit));


// Return if no parameter is remaining...
IF ( ParameterCnt = 0 ) THEN RETURN; END_IF
// dec remaining parameter(s)                        
ParameterCnt := ParameterCnt - 1;
// Create log entry for WorkAreaData.E4Limit.LowerLimit
CreateLogMessagePara1 ( Timestamp   := Timestamp,
                        MessageType := MessageType.CMD,
                        Severity    := Severity.DEBUG,
                        MessageCode := 0,
                        MessageText := 'Response.WorkAreaData.E4Limit.LowerLimit = {1}',
                        Para1       :=  REAL_TO_STRING(_response.WorkAreaData.E4Limit.LowerLimit));


// Return if no parameter is remaining...
IF ( ParameterCnt = 0 ) THEN RETURN; END_IF
// dec remaining parameter(s)                        
ParameterCnt := ParameterCnt - 1;
// Create log entry for WorkAreaData.E5Limit.LowerLimit
CreateLogMessagePara1 ( Timestamp   := Timestamp,
                        MessageType := MessageType.CMD,
                        Severity    := Severity.DEBUG,
                        MessageCode := 0,
                        MessageText := 'Response.WorkAreaData.E5Limit.LowerLimit = {1}',
                        Para1       :=  REAL_TO_STRING(_response.WorkAreaData.E5Limit.LowerLimit));


// Return if no parameter is remaining...
IF ( ParameterCnt = 0 ) THEN RETURN; END_IF
// dec remaining parameter(s)                        
ParameterCnt := ParameterCnt - 1;
// Create log entry for WorkAreaData.E6Limit.LowerLimit
CreateLogMessagePara1 ( Timestamp   := Timestamp,
                        MessageType := MessageType.CMD,
                        Severity    := Severity.DEBUG,
                        MessageCode := 0,
                        MessageText := 'Response.WorkAreaData.E6Limit.LowerLimit = {1}',
                        Para1       :=  REAL_TO_STRING(_response.WorkAreaData.E6Limit.LowerLimit));


// Return if no parameter is remaining...
IF ( ParameterCnt = 0 ) THEN RETURN; END_IF
// dec remaining parameter(s)                        
ParameterCnt := ParameterCnt - 1;
// Create log entry for WorkAreaData.E2Limit.UpperLimit
CreateLogMessagePara1 ( Timestamp   := Timestamp,
                        MessageType := MessageType.CMD,
                        Severity    := Severity.DEBUG,
                        MessageCode := 0,
                        MessageText := 'Response.WorkAreaData.E2Limit.UpperLimit = {1}',
                        Para1       :=  REAL_TO_STRING(_response.WorkAreaData.E2Limit.UpperLimit));


// Return if no parameter is remaining...
IF ( ParameterCnt = 0 ) THEN RETURN; END_IF
// dec remaining parameter(s)                        
ParameterCnt := ParameterCnt - 1;
// Create log entry for WorkAreaData.E3Limit.UpperLimit
CreateLogMessagePara1 ( Timestamp   := Timestamp,
                        MessageType := MessageType.CMD,
                        Severity    := Severity.DEBUG,
                        MessageCode := 0,
                        MessageText := 'Response.WorkAreaData.E3Limit.UpperLimit = {1}',
                        Para1       :=  REAL_TO_STRING(_response.WorkAreaData.E3Limit.UpperLimit));


// Return if no parameter is remaining...
IF ( ParameterCnt = 0 ) THEN RETURN; END_IF
// dec remaining parameter(s)                        
ParameterCnt := ParameterCnt - 1;
// Create log entry for WorkAreaData.E4Limit.UpperLimit
CreateLogMessagePara1 ( Timestamp   := Timestamp,
                        MessageType := MessageType.CMD,
                        Severity    := Severity.DEBUG,
                        MessageCode := 0,
                        MessageText := 'Response.WorkAreaData.E4Limit.UpperLimit = {1}',
                        Para1       :=  REAL_TO_STRING(_response.WorkAreaData.E4Limit.UpperLimit));


// Return if no parameter is remaining...
IF ( ParameterCnt = 0 ) THEN RETURN; END_IF
// dec remaining parameter(s)                        
ParameterCnt := ParameterCnt - 1;
// Create log entry for WorkAreaData.E5Limit.UpperLimit
CreateLogMessagePara1 ( Timestamp   := Timestamp,
                        MessageType := MessageType.CMD,
                        Severity    := Severity.DEBUG,
                        MessageCode := 0,
                        MessageText := 'Response.WorkAreaData.E5Limit.UpperLimit = {1}',
                        Para1       :=  REAL_TO_STRING(_response.WorkAreaData.E5Limit.UpperLimit));


// Return if no parameter is remaining...
IF ( ParameterCnt = 0 ) THEN RETURN; END_IF
// dec remaining parameter(s)                        
ParameterCnt := ParameterCnt - 1;
// Create log entry for WorkAreaData.E6Limit.UpperLimit
CreateLogMessagePara1 ( Timestamp   := Timestamp,
                        MessageType := MessageType.CMD,
                        Severity    := Severity.DEBUG,
                        MessageCode := 0,
                        MessageText := 'Response.WorkAreaData.E6Limit.UpperLimit = {1}',
                        Para1       :=  REAL_TO_STRING(_response.WorkAreaData.E6Limit.UpperLimit));
                
END_METHOD

METHOD PROTECTED Reset : DINT
VAR_INPUT
END_VAR
                  Reset := SUPER^.Reset();

Done               := FALSE;
Busy               := FALSE;
CommandBuffered    := FALSE;
                
END_METHOD
END_FUNCTION_BLOCK

/// Define work area
FUNCTION_BLOCK MC_WriteWorkAreaFB EXTENDS RobotLibraryBaseExecuteFB
// ------------------------------------------------------------------------- 
//  SRCI Robot Library                                                
// ------------------------------------------------------------------------- 
//                                                                           
//  Object:      WriteWorkAreaFB                                       
//  Author:      Thorsten Brach                                                
//  Date:        2024-06-01
//
//  Description:                                              
//   
//                                                                           
//  Copyright: 
//    (C) 2024 Thorsten Brach. All rights reserved                                                                                                                                            
//             Licensed under the MIT License.
//                                                                           
//  Disclaimer:                                                                           
//    This project is provided without any guarantee and can be used for   
//    private and commercial purposes. Any use is at the user’s 
//    own risk and responsibility.
//
// -------------------------------------------------------------------------
VAR_INPUT
  /// Processing Mode
  ProcessingMode     : ProcessingMode;
  /// command parameter 
  ParCmd             : WriteWorkAreaParCmd;
END_VAR
VAR_OUTPUT
  /// Command is transferred and confirmed by the RC
  CommandBuffered    : BOOL;
  /// command outputs
  OutCmd             : WriteWorkAreaOutCmd;       
END_VAR

VAR
  /// internal copy of command parameter 
 _parCmd             : WriteWorkAreaParCmd;
  /// command data to send
 _command            : WriteWorkAreaSendData;
  /// response data received
 _response           : WriteWorkAreaRecvData;      
END_VAR

            SUPER^(AxesGroup := AxesGroup);
          

METHOD INTERNAL CheckAddParameter : BOOL
VAR_INPUT
  /// Payload pointer
  PayloadPtr : UDINT;
END_VAR
VAR
  /// Payload as byte array
  Payload    : ARRAY [1..SIZEOF(_command)] OF BYTE;
  /// Null Byte array 
  Null       : ARRAY [1..SIZEOF(_command)] OF BYTE;
  /// Data length to compare
  DataLen    : UDINT;
END_VAR
                  // Payload pointer must be decreased by one byte, because ADR(Payload) is already one byte !
PayloadPtr := LIMIT (0, PayloadPtr - 1, SIZEOF(Payload) -1);
// Convert command struct to payload array
SysDepMemCpy( pDest := ADR(Payload), pSrc := ADR(_command), DataLen := SIZEOF(_command));
// Calculate the data length to compare - at least one byte must be compared !
DataLen := LIMIT(1, SIZEOF(Payload) - PayloadPtr, SIZEOF(Payload)); 
// Compare Payload-Array with Null-Byte-Array
CheckAddParameter := SysDepMemCmp( pData1 := ADR(Payload) + PayloadPtr , pData2 := ADR(Null), DataLen := DataLen) <>  RobotLibraryConstants.OK ;
                
END_METHOD

METHOD PROTECTED CheckFunctionSupported : BOOL
VAR_IN_OUT
  /// Robot assignment of function
  AxesGroup : AxesGroup; 
END_VAR
                  CheckFunctionSupported := AxesGroup.State.RobotData.RCSupportedFunctions.WriteWorkArea;

IF ( NOT CheckFunctionSupported )
THEN
  // call base implementation for set error and create log entry
  SUPER^.CheckFunctionSupported(AxesGroup := AxesGroup);
END_IF
                
END_METHOD

METHOD PROTECTED CheckParameterChanged : BOOL
VAR_IN_OUT
  /// Robot assignment of function
  AxesGroup    : AxesGroup; 
END_VAR
                  // Check ParCmd Size is > 0, because MemCmp does not work correctly with size = 0
IF (SIZEOF(ParCmd) = 0) OR (_stepCmd = 0)
THEN 
  RETURN;
END_IF

// compare memory 
_parameterChanged := ( SysDepMemCmp(pData1 := ADR(ParCmd), pData2 := ADR(_parCmd), DataLen := SIZEOF(ParCmd)) <> RobotLibraryConstants.OK );

// check parameter valid ?
_parameterValid   := CheckParameterValid( AxesGroup := AxesGroup );

IF ((  _parameterChanged        )  AND 
    (  _parameterValid          )) OR
    (  _parameterUpdateInternal )  
THEN  
  // Create log entry for parameter changed event
  CreateLogMessagePara1 ( Timestamp   := AxesGroup.State.SystemTime,
                          MessageType := MessageType.CMD,
                          Severity    := Severity.DEBUG,
                          MessageCode := 0,
                          MessageText := 'NotifyParameterChanged Event {1}',
                          Para1       :=  '' );

  // reset internal flag for send parameter update
 _parameterUpdateInternal := FALSE;
  // update internal copy of parameters 
 _parCmd := ParCmd;
  // inc parameter sequence
 _command.ParSeq := _command.ParSeq + 1;
  // update command data  
  CommandData := CreateCommandPayload(AxesGroup := AxesGroup); // ( Access via reference to rCommandFB in ACR )
  // notify active command register 
  AxesGroup.Acyclic.ActiveCommandRegister.NotifyParameterChanged := _uniqueID;
END_IF
                
END_METHOD

METHOD PROTECTED CheckParameterValid : BOOL
VAR_IN_OUT
  /// Robot assignment of function
  AxesGroup : AxesGroup; 
END_VAR
VAR
  /// internal index for loops
 _idx : DINT;
END_VAR
                  CheckParameterValid := TRUE;


// Check ParCmd.WorkAreaNo valid ? 
IF (( ParCmd.WorkAreaNo < 0                                                      ) OR  
    ( ParCmd.WorkAreaNo > 254                                                    ) OR
    ( ParCmd.WorkAreaNo > AxesGroup.State.ConfigurationData.HighestWorkAreaIndex ) OR
    ( ParCmd.WorkAreaNo > AxesGroup.State.UnifiedWorkAreaIndex                   ))         
THEN
  // Parameter not valid
  CheckParameterValid := FALSE;
  
  // Check LoadNo available on RC ? 
  IF ( ParCmd.WorkAreaNo > AxesGroup.State.ConfigurationData.HighestWorkAreaIndex )
  THEN
    SetError( ErrorID := RobotLibraryErrorIdEnum.ERR_WORKAREANO_UNAVAILABLE, Overwrite := TRUE );
  ELSE
    SetError( ErrorID := RobotLibraryErrorIdEnum.ERR_WORKAREANO_RANGE, Overwrite := TRUE );
	END_IF  
  
  // Create log entry
  CreateLogMessagePara1 ( Timestamp   := AxesGroup.State.SystemTime,
                          MessageType := MessageType.CMD,
                          Severity    := Severity.ERROR,
                          MessageCode := ErrorID,
                          MessageText := 'Invalid Parameter ParCmd.WorkAreaNo = {1}',
                          Para1       := USINT_TO_STRING(ParCmd.WorkAreaNo));
  RETURN;
END_IF


// Check ParCmd.WorkAreaData.AreaType valid ? 
IF (( ParCmd.WorkAreaData.AreaType <> AreaType.AXES     ) AND
    ( ParCmd.WorkAreaData.AreaType <> AreaType.BOX      ) AND
    ( ParCmd.WorkAreaData.AreaType <> AreaType.CYLINDER ) AND
    ( ParCmd.WorkAreaData.AreaType <> AreaType.SPHERE   ))
THEN
  // Parameter not valid
  CheckParameterValid := FALSE;
  // Set error
  SetError( ErrorID := RobotLibraryErrorIdEnum.ERR_INVALID_PAR_CMD, Overwrite := TRUE );
  // Create log entry
  CreateLogMessagePara1 ( Timestamp   := AxesGroup.State.SystemTime,
                          MessageType := MessageType.CMD,
                          Severity    := Severity.ERROR,
                          MessageCode := ErrorID,
                          MessageText := 'Invalid Parameter ParCmd.WorkAreaData.AreaType = {1}',
                          Para1       := AREA_TYPE_TO_STRING(ParCmd.WorkAreaData.AreaType));
  RETURN;
END_IF


// Check ParCmd.WorkAreaData.AreaMode valid ? 
IF (( ParCmd.WorkAreaData.AreaMode <> FALSE ) AND
    ( ParCmd.WorkAreaData.AreaMode <> TRUE  ))
THEN
  // Parameter not valid
  CheckParameterValid := FALSE;
  // Set error
  SetError( ErrorID := RobotLibraryErrorIdEnum.ERR_INVALID_PAR_CMD, Overwrite := TRUE );
  // Create log entry
  CreateLogMessagePara1 ( Timestamp   := AxesGroup.State.SystemTime,
                          MessageType := MessageType.CMD,
                          Severity    := Severity.ERROR,
                          MessageCode := ErrorID,
                          MessageText := 'Invalid Parameter ParCmd.WorkAreaData.AreaMode = {1}',
                          Para1       := BOOL_TO_STRING(ParCmd.WorkAreaData.AreaMode));
  RETURN;
END_IF


// Check ParCmd.WorkAreaData.ReactionMode valid ? 
IF (( ParCmd.WorkAreaData.ReactionMode <> WorkAreaReactionMode.NO_REACTION ) AND
    ( ParCmd.WorkAreaData.ReactionMode <> WorkAreaReactionMode.ABORT       ) AND
    ( ParCmd.WorkAreaData.ReactionMode <> WorkAreaReactionMode.INTERRUPT   ))
THEN
  // Parameter not valid
  CheckParameterValid := FALSE;
  // Set error
  SetError( ErrorID := RobotLibraryErrorIdEnum.ERR_INVALID_PAR_CMD, Overwrite := TRUE );
  // Create log entry
  CreateLogMessagePara1 ( Timestamp   := AxesGroup.State.SystemTime,
                          MessageType := MessageType.CMD,
                          Severity    := Severity.ERROR,
                          MessageCode := ErrorID,
                          MessageText := 'Invalid Parameter ParCmd.WorkAreaData.ReactionMode = {1}',
                          Para1       := WORK_AREA_REACTION_MODE_TO_STRING(ParCmd.WorkAreaData.ReactionMode));
  RETURN;
END_IF


// Check ParCmd.WorkAreaData.ActiveModification valid ? 
IF (( ParCmd.WorkAreaData.ActiveModification <> FALSE ) AND
    ( ParCmd.WorkAreaData.ActiveModification <> TRUE  ))
THEN
  // Parameter not valid
  CheckParameterValid := FALSE;
  // Set error
  SetError( ErrorID := RobotLibraryErrorIdEnum.ERR_INVALID_PAR_CMD, Overwrite := TRUE );
  // Create log entry
  CreateLogMessagePara1 ( Timestamp   := AxesGroup.State.SystemTime,
                          MessageType := MessageType.CMD,
                          Severity    := Severity.ERROR,
                          MessageCode := ErrorID,
                          MessageText := 'Invalid Parameter ParCmd.WorkAreaData.ActiveModification = {1}',
                          Para1       := BOOL_TO_STRING(ParCmd.WorkAreaData.ActiveModification));
  RETURN;
END_IF


// Check ParCmd.WorkAreaData.DefinitionMode valid ? 
IF (( ParCmd.WorkAreaData.DefinitionMode <> DefinitionMode.Center ) AND
    ( ParCmd.WorkAreaData.DefinitionMode <> DefinitionMode.Face   ))
THEN
  // Parameter not valid
  CheckParameterValid := FALSE;
  // Set error
  SetError( ErrorID := RobotLibraryErrorIdEnum.ERR_INVALID_PAR_CMD, Overwrite := TRUE );
  // Create log entry
  CreateLogMessagePara1 ( Timestamp   := AxesGroup.State.SystemTime,
                          MessageType := MessageType.CMD,
                          Severity    := Severity.ERROR,
                          MessageCode := ErrorID,
                          MessageText := 'Invalid Parameter ParCmd.WorkAreaData.DefinitionMode = {1}',
                          Para1       := DEFINITION_MODE_TO_STRING(ParCmd.WorkAreaData.DefinitionMode));
  RETURN;
END_IF


// Check ParCmd.WorkAreaData.FrameNo valid ? 
IF (( ParCmd.WorkAreaData.FrameNo < 0   ) OR
    ( ParCmd.WorkAreaData.FrameNo> 254 ))
      
THEN
  // Parameter not valid
  CheckParameterValid := FALSE;
  // Set error
  SetError( ErrorID := RobotLibraryErrorIdEnum.ERR_INVALID_PAR_CMD, Overwrite := TRUE );
  // Create log entry
  CreateLogMessagePara1 ( Timestamp   := AxesGroup.State.SystemTime,
                          MessageType := MessageType.CMD,
                          Severity    := Severity.ERROR,
                          MessageCode := ErrorID,
                          MessageText := 'Invalid Parameter ParCmd.WorkAreaData.FrameNo = {1}',
                          Para1       := USINT_TO_STRING(ParCmd.WorkAreaData.FrameNo));
  RETURN;
END_IF


// Check ParCmd.WorkAreaData.ZeroPointX valid ? 
IF ( SysDepIsValidReal(ParCmd.WorkAreaData.ZeroPointX) = FALSE ) 
THEN
  // Parameter not valid
  CheckParameterValid := FALSE;
  // Set error
  SetError( ErrorID := RobotLibraryErrorIdEnum.ERR_INVALID_PAR_CMD, Overwrite := TRUE );
  
  // Create log entry
  CreateLogMessagePara1 ( Timestamp   := AxesGroup.State.SystemTime,
                          MessageType := MessageType.CMD,
                          Severity    := Severity.ERROR,
                          MessageCode := ErrorID,
                          MessageText := 'Invalid Parameter ParCmd.WorkAreaData.ZeroPointX = {1}',
                          Para1       := VALID_REAL_TO_STRING(ParCmd.WorkAreaData.ZeroPointX));
  RETURN;                          
END_IF


// Check ParCmd.WorkAreaData.ZeroPointY valid ? 
IF ( SysDepIsValidReal(ParCmd.WorkAreaData.ZeroPointY) = FALSE ) 
THEN
  // Parameter not valid
  CheckParameterValid := FALSE;
  // Set error
  SetError( ErrorID := RobotLibraryErrorIdEnum.ERR_INVALID_PAR_CMD, Overwrite := TRUE );
  
  // Create log entry
  CreateLogMessagePara1 ( Timestamp   := AxesGroup.State.SystemTime,
                          MessageType := MessageType.CMD,
                          Severity    := Severity.ERROR,
                          MessageCode := ErrorID,
                          MessageText := 'Invalid Parameter ParCmd.WorkAreaData.ZeroPointY = {1}',
                          Para1       := VALID_REAL_TO_STRING(ParCmd.WorkAreaData.ZeroPointY));
  RETURN;                          
END_IF


// Check ParCmd.WorkAreaData.ZeroPointZ valid ? 
IF ( SysDepIsValidReal(ParCmd.WorkAreaData.ZeroPointZ) = FALSE ) 
THEN
  // Parameter not valid
  CheckParameterValid := FALSE;
  // Set error
  SetError( ErrorID := RobotLibraryErrorIdEnum.ERR_INVALID_PAR_CMD, Overwrite := TRUE );
  
  // Create log entry
  CreateLogMessagePara1 ( Timestamp   := AxesGroup.State.SystemTime,
                          MessageType := MessageType.CMD,
                          Severity    := Severity.ERROR,
                          MessageCode := ErrorID,
                          MessageText := 'Invalid Parameter ParCmd.WorkAreaData.ZeroPointZ = {1}',
                          Para1       := VALID_REAL_TO_STRING(ParCmd.WorkAreaData.ZeroPointZ));
  RETURN;                          
END_IF


// Check ParCmd.WorkAreaData.X.LowerLimit ? 
IF ( SysDepIsValidReal(ParCmd.WorkAreaData.X.LowerLimit) = FALSE ) 
THEN
  // Parameter not valid
  CheckParameterValid := FALSE;
  // Set error
  SetError( ErrorID := RobotLibraryErrorIdEnum.ERR_INVALID_PAR_CMD, Overwrite := TRUE );
  
  // Create log entry
  CreateLogMessagePara1 ( Timestamp   := AxesGroup.State.SystemTime,
                          MessageType := MessageType.CMD,
                          Severity    := Severity.ERROR,
                          MessageCode := ErrorID,
                          MessageText := 'Invalid Parameter ParCmd.WorkAreaData.X.LowerLimit = {1}',
                          Para1       := VALID_REAL_TO_STRING(ParCmd.WorkAreaData.X.LowerLimit));
  RETURN;                          
END_IF


// Check ParCmd.WorkAreaData.X.UpperLimit ? 
IF ( SysDepIsValidReal(ParCmd.WorkAreaData.X.UpperLimit) = FALSE ) 
THEN
  // Parameter not valid
  CheckParameterValid := FALSE;
  // Set error
  SetError( ErrorID := RobotLibraryErrorIdEnum.ERR_INVALID_PAR_CMD, Overwrite := TRUE );
  
  // Create log entry
  CreateLogMessagePara1 ( Timestamp   := AxesGroup.State.SystemTime,
                          MessageType := MessageType.CMD,
                          Severity    := Severity.ERROR,
                          MessageCode := ErrorID,
                          MessageText := 'Invalid Parameter ParCmd.WorkAreaData.X.UpperLimit = {1}',
                          Para1       := VALID_REAL_TO_STRING(ParCmd.WorkAreaData.X.UpperLimit));
  RETURN;                          
END_IF


// Check ParCmd.WorkAreaData.Y.LowerLimit ? 
IF ( SysDepIsValidReal(ParCmd.WorkAreaData.Y.LowerLimit) = FALSE ) 
THEN
  // Parameter not valid
  CheckParameterValid := FALSE;
  // Set error
  SetError( ErrorID := RobotLibraryErrorIdEnum.ERR_INVALID_PAR_CMD, Overwrite := TRUE );
  
  // Create log entry
  CreateLogMessagePara1 ( Timestamp   := AxesGroup.State.SystemTime,
                          MessageType := MessageType.CMD,
                          Severity    := Severity.ERROR,
                          MessageCode := ErrorID,
                          MessageText := 'Invalid Parameter ParCmd.WorkAreaData.Y.LowerLimit = {1}',
                          Para1       := VALID_REAL_TO_STRING(ParCmd.WorkAreaData.Y.LowerLimit));
  RETURN;                          
END_IF


// Check ParCmd.WorkAreaData.Y.UpperLimit ? 
IF ( SysDepIsValidReal(ParCmd.WorkAreaData.Y.UpperLimit) = FALSE ) 
THEN
  // Parameter not valid
  CheckParameterValid := FALSE;
  // Set error
  SetError( ErrorID := RobotLibraryErrorIdEnum.ERR_INVALID_PAR_CMD, Overwrite := TRUE );
  
  // Create log entry
  CreateLogMessagePara1 ( Timestamp   := AxesGroup.State.SystemTime,
                          MessageType := MessageType.CMD,
                          Severity    := Severity.ERROR,
                          MessageCode := ErrorID,
                          MessageText := 'Invalid Parameter ParCmd.WorkAreaData.Y.UpperLimit = {1}',
                          Para1       := VALID_REAL_TO_STRING(ParCmd.WorkAreaData.Y.UpperLimit));
  RETURN;                          
END_IF


// Check ParCmd.WorkAreaData.Z.LowerLimit ? 
IF ( SysDepIsValidReal(ParCmd.WorkAreaData.Z.LowerLimit) = FALSE ) 
THEN
  // Parameter not valid
  CheckParameterValid := FALSE;
  // Set error
  SetError( ErrorID := RobotLibraryErrorIdEnum.ERR_INVALID_PAR_CMD, Overwrite := TRUE );
  
  // Create log entry
  CreateLogMessagePara1 ( Timestamp   := AxesGroup.State.SystemTime,
                          MessageType := MessageType.CMD,
                          Severity    := Severity.ERROR,
                          MessageCode := ErrorID,
                          MessageText := 'Invalid Parameter ParCmd.WorkAreaData.Z.LowerLimit = {1}',
                          Para1       := VALID_REAL_TO_STRING(ParCmd.WorkAreaData.Z.LowerLimit));
  RETURN;                          
END_IF

// Check ParCmd.WorkAreaData.Z.UpperLimit ? 
IF ( SysDepIsValidReal(ParCmd.WorkAreaData.Z.UpperLimit) = FALSE ) 
THEN
  // Parameter not valid
  CheckParameterValid := FALSE;
  // Set error
  SetError( ErrorID := RobotLibraryErrorIdEnum.ERR_INVALID_PAR_CMD, Overwrite := TRUE );
  
  // Create log entry
  CreateLogMessagePara1 ( Timestamp   := AxesGroup.State.SystemTime,
                          MessageType := MessageType.CMD,
                          Severity    := Severity.ERROR,
                          MessageCode := ErrorID,
                          MessageText := 'Invalid Parameter ParCmd.WorkAreaData.Z.UpperLimit = {1}',
                          Para1       := VALID_REAL_TO_STRING(ParCmd.WorkAreaData.Z.UpperLimit));
  RETURN;                          
END_IF


// Check ParCmd.WorkAreaData.Radius ? 
IF ( SysDepIsValidReal(ParCmd.WorkAreaData.Radius) = FALSE ) 
THEN
  // Parameter not valid
  CheckParameterValid := FALSE;
  // Set error
  SetError( ErrorID := RobotLibraryErrorIdEnum.ERR_INVALID_PAR_CMD, Overwrite := TRUE );
  
  // Create log entry
  CreateLogMessagePara1 ( Timestamp   := AxesGroup.State.SystemTime,
                          MessageType := MessageType.CMD,
                          Severity    := Severity.ERROR,
                          MessageCode := ErrorID,
                          MessageText := 'Invalid Parameter ParCmd.Radius = {1}',
                          Para1       := VALID_REAL_TO_STRING(ParCmd.WorkAreaData.Radius));
  RETURN;                          
END_IF


// Check ParCmd.WorkAreaData.J1Limit.LowerLimit ? 
IF ( SysDepIsValidReal(ParCmd.WorkAreaData.J1Limit.LowerLimit) = FALSE ) 
THEN
  // Parameter not valid
  CheckParameterValid := FALSE;
  // Set error
  SetError( ErrorID := RobotLibraryErrorIdEnum.ERR_INVALID_PAR_CMD, Overwrite := TRUE );
  
  // Create log entry
  CreateLogMessagePara1 ( Timestamp   := AxesGroup.State.SystemTime,
                          MessageType := MessageType.CMD,
                          Severity    := Severity.ERROR,
                          MessageCode := ErrorID,
                          MessageText := 'Invalid Parameter ParCmd.J1Limit.LowerLimit = {1}',
                          Para1       := VALID_REAL_TO_STRING(ParCmd.WorkAreaData.J1Limit.LowerLimit));
  RETURN;                          
END_IF


// Check ParCmd.WorkAreaData.J1Limit.UpperLimit ? 
IF ( SysDepIsValidReal(ParCmd.WorkAreaData.J1Limit.UpperLimit) = FALSE ) 
THEN
  // Parameter not valid
  CheckParameterValid := FALSE;
  // Set error
  SetError( ErrorID := RobotLibraryErrorIdEnum.ERR_INVALID_PAR_CMD, Overwrite := TRUE );
  
  // Create log entry
  CreateLogMessagePara1 ( Timestamp   := AxesGroup.State.SystemTime,
                          MessageType := MessageType.CMD,
                          Severity    := Severity.ERROR,
                          MessageCode := ErrorID,
                          MessageText := 'Invalid Parameter ParCmd.J1Limit.UpperLimit = {1}',
                          Para1       := VALID_REAL_TO_STRING(ParCmd.WorkAreaData.J1Limit.UpperLimit));
  RETURN;                          
END_IF


// Check ParCmd.WorkAreaData.J2Limit.LowerLimit ? 
IF ( SysDepIsValidReal(ParCmd.WorkAreaData.J2Limit.LowerLimit) = FALSE ) 
THEN
  // Parameter not valid
  CheckParameterValid := FALSE;
  // Set error
  SetError( ErrorID := RobotLibraryErrorIdEnum.ERR_INVALID_PAR_CMD, Overwrite := TRUE );
  
  // Create log entry
  CreateLogMessagePara1 ( Timestamp   := AxesGroup.State.SystemTime,
                          MessageType := MessageType.CMD,
                          Severity    := Severity.ERROR,
                          MessageCode := ErrorID,
                          MessageText := 'Invalid Parameter ParCmd.J2Limit.LowerLimit = {1}',
                          Para1       := VALID_REAL_TO_STRING(ParCmd.WorkAreaData.J2Limit.LowerLimit));
  RETURN;                          
END_IF


// Check ParCmd.WorkAreaData.J2Limit.UpperLimit ? 
IF ( SysDepIsValidReal(ParCmd.WorkAreaData.J2Limit.UpperLimit) = FALSE ) 
THEN
  // Parameter not valid
  CheckParameterValid := FALSE;
  // Set error
  SetError( ErrorID := RobotLibraryErrorIdEnum.ERR_INVALID_PAR_CMD, Overwrite := TRUE );
  
  // Create log entry
  CreateLogMessagePara1 ( Timestamp   := AxesGroup.State.SystemTime,
                          MessageType := MessageType.CMD,
                          Severity    := Severity.ERROR,
                          MessageCode := ErrorID,
                          MessageText := 'Invalid Parameter ParCmd.J2Limit.UpperLimit = {1}',
                          Para1       := VALID_REAL_TO_STRING(ParCmd.WorkAreaData.J2Limit.UpperLimit));
  RETURN;                          
END_IF


// Check ParCmd.WorkAreaData.J3Limit.LowerLimit ? 
IF ( SysDepIsValidReal(ParCmd.WorkAreaData.J3Limit.LowerLimit) = FALSE ) 
THEN
  // Parameter not valid
  CheckParameterValid := FALSE;
  // Set error
  SetError( ErrorID := RobotLibraryErrorIdEnum.ERR_INVALID_PAR_CMD, Overwrite := TRUE );
  
  // Create log entry
  CreateLogMessagePara1 ( Timestamp   := AxesGroup.State.SystemTime,
                          MessageType := MessageType.CMD,
                          Severity    := Severity.ERROR,
                          MessageCode := ErrorID,
                          MessageText := 'Invalid Parameter ParCmd.J3Limit.LowerLimit = {1}',
                          Para1       := VALID_REAL_TO_STRING(ParCmd.WorkAreaData.J3Limit.LowerLimit));
  RETURN;                          
END_IF


// Check ParCmd.WorkAreaData.J3Limit.UpperLimit ? 
IF ( SysDepIsValidReal(ParCmd.WorkAreaData.J3Limit.UpperLimit) = FALSE ) 
THEN
  // Parameter not valid
  CheckParameterValid := FALSE;
  // Set error
  SetError( ErrorID := RobotLibraryErrorIdEnum.ERR_INVALID_PAR_CMD, Overwrite := TRUE );
  
  // Create log entry
  CreateLogMessagePara1 ( Timestamp   := AxesGroup.State.SystemTime,
                          MessageType := MessageType.CMD,
                          Severity    := Severity.ERROR,
                          MessageCode := ErrorID,
                          MessageText := 'Invalid Parameter ParCmd.J3Limit.UpperLimit = {1}',
                          Para1       := VALID_REAL_TO_STRING(ParCmd.WorkAreaData.J3Limit.UpperLimit));
  RETURN;                          
END_IF


// Check ParCmd.WorkAreaData.J4Limit.LowerLimit ? 
IF ( SysDepIsValidReal(ParCmd.WorkAreaData.J4Limit.LowerLimit) = FALSE ) 
THEN
  // Parameter not valid
  CheckParameterValid := FALSE;
  // Set error
  SetError( ErrorID := RobotLibraryErrorIdEnum.ERR_INVALID_PAR_CMD, Overwrite := TRUE );
  
  // Create log entry
  CreateLogMessagePara1 ( Timestamp   := AxesGroup.State.SystemTime,
                          MessageType := MessageType.CMD,
                          Severity    := Severity.ERROR,
                          MessageCode := ErrorID,
                          MessageText := 'Invalid Parameter ParCmd.J4Limit.LowerLimit = {1}',
                          Para1       := VALID_REAL_TO_STRING(ParCmd.WorkAreaData.J4Limit.LowerLimit));
  RETURN;                          
END_IF


// Check ParCmd.WorkAreaData.J4Limit.UpperLimit ? 
IF ( SysDepIsValidReal(ParCmd.WorkAreaData.J4Limit.UpperLimit) = FALSE ) 
THEN
  // Parameter not valid
  CheckParameterValid := FALSE;
  // Set error
  SetError( ErrorID := RobotLibraryErrorIdEnum.ERR_INVALID_PAR_CMD, Overwrite := TRUE );
  
  // Create log entry
  CreateLogMessagePara1 ( Timestamp   := AxesGroup.State.SystemTime,
                          MessageType := MessageType.CMD,
                          Severity    := Severity.ERROR,
                          MessageCode := ErrorID,
                          MessageText := 'Invalid Parameter ParCmd.J4Limit.UpperLimit = {1}',
                          Para1       := VALID_REAL_TO_STRING(ParCmd.WorkAreaData.J4Limit.UpperLimit));
  RETURN;                          
END_IF


// Check ParCmd.WorkAreaData.J5Limit.LowerLimit ? 
IF ( SysDepIsValidReal(ParCmd.WorkAreaData.J5Limit.LowerLimit) = FALSE ) 
THEN
  // Parameter not valid
  CheckParameterValid := FALSE;
  // Set error
  SetError( ErrorID := RobotLibraryErrorIdEnum.ERR_INVALID_PAR_CMD, Overwrite := TRUE );
  
  // Create log entry
  CreateLogMessagePara1 ( Timestamp   := AxesGroup.State.SystemTime,
                          MessageType := MessageType.CMD,
                          Severity    := Severity.ERROR,
                          MessageCode := ErrorID,
                          MessageText := 'Invalid Parameter ParCmd.J5Limit.LowerLimit = {1}',
                          Para1       := VALID_REAL_TO_STRING(ParCmd.WorkAreaData.J5Limit.LowerLimit));
  RETURN;                          
END_IF


// Check ParCmd.WorkAreaData.J5Limit.UpperLimit ? 
IF ( SysDepIsValidReal(ParCmd.WorkAreaData.J5Limit.UpperLimit) = FALSE ) 
THEN
  // Parameter not valid
  CheckParameterValid := FALSE;
  // Set error
  SetError( ErrorID := RobotLibraryErrorIdEnum.ERR_INVALID_PAR_CMD, Overwrite := TRUE );
  
  // Create log entry
  CreateLogMessagePara1 ( Timestamp   := AxesGroup.State.SystemTime,
                          MessageType := MessageType.CMD,
                          Severity    := Severity.ERROR,
                          MessageCode := ErrorID,
                          MessageText := 'Invalid Parameter ParCmd.J5Limit.UpperLimit = {1}',
                          Para1       := VALID_REAL_TO_STRING(ParCmd.WorkAreaData.J5Limit.UpperLimit));
  RETURN;                          
END_IF


// Check ParCmd.WorkAreaData.J6Limit.LowerLimit ? 
IF ( SysDepIsValidReal(ParCmd.WorkAreaData.J6Limit.LowerLimit) = FALSE ) 
THEN
  // Parameter not valid
  CheckParameterValid := FALSE;
  // Set error
  SetError( ErrorID := RobotLibraryErrorIdEnum.ERR_INVALID_PAR_CMD, Overwrite := TRUE );
  
  // Create log entry
  CreateLogMessagePara1 ( Timestamp   := AxesGroup.State.SystemTime,
                          MessageType := MessageType.CMD,
                          Severity    := Severity.ERROR,
                          MessageCode := ErrorID,
                          MessageText := 'Invalid Parameter ParCmd.J6Limit.LowerLimit = {1}',
                          Para1       := VALID_REAL_TO_STRING(ParCmd.WorkAreaData.J6Limit.LowerLimit));
  RETURN;                          
END_IF


// Check ParCmd.WorkAreaData.J6Limit.UpperLimit ? 
IF ( SysDepIsValidReal(ParCmd.WorkAreaData.J6Limit.UpperLimit) = FALSE ) 
THEN
  // Parameter not valid
  CheckParameterValid := FALSE;
  // Set error
  SetError( ErrorID := RobotLibraryErrorIdEnum.ERR_INVALID_PAR_CMD, Overwrite := TRUE );
  
  // Create log entry
  CreateLogMessagePara1 ( Timestamp   := AxesGroup.State.SystemTime,
                          MessageType := MessageType.CMD,
                          Severity    := Severity.ERROR,
                          MessageCode := ErrorID,
                          MessageText := 'Invalid Parameter ParCmd.J6Limit.UpperLimit = {1}',
                          Para1       := VALID_REAL_TO_STRING(ParCmd.WorkAreaData.J6Limit.UpperLimit));
  RETURN;                          
END_IF
                
END_METHOD

METHOD INTERNAL CreateCommandPayload : RobotLibraryCommandDataFB
VAR_IN_OUT
  /// Robot assignment of function
  AxesGroup : AxesGroup; 
END_VAR
VAR
  /// Parameter count
 _parameterCnt : DINT;
END_VAR
// Table 6-205: Sent CMD payload (PLC to RC) of "WriteWorkArea"
// --------------------------
// Header
// --------------------------
// Byte 00 : UINT  - Type HB     
// Byte 01 :       - Type LB    
// Byte 02 : USINT - Reserve | ExecutionMode
// Byte 03 : USINT - ParSeq  | Priority
// --------------------------
// Datablock
// --------------------------
// Byte 04 : UINT WorkAreaNo
// Byte 05 : 
// Byte 06 : DATE Data.Date
// Byte 07 : 
// Byte 08 : TIME_OF_DAY Data.Time
// Byte 09 : 
// Byte 10 : 
// Byte 11 : USINT - Data.AreaType
// Byte 12 : BOOL  - Data.AreaMode
// Byte 13 : USINT - Data.ReactionMode
// Byte 14 : BOOL  - Data.ActiveModification
// Byte 15 : USINT - Data.DefinitionMode
// Byte 16 : USINT - Data.FrameNo
// Byte 17 : 
// Byte 18 : REAL  - Data.ZeroPointX
// Byte 19 : 
// Byte 20 : 
// Byte 21 : 
// Byte 22 : REAL  - Data.ZeroPointY
// Byte 23 : 
// Byte 24 : 
// Byte 25 : 
// Byte 26 : REAL  - Data.ZeroPointZ
// Byte 27 : 
// Byte 28 : 
// Byte 29 : 
// Byte 30 : REAL  - Data.X1
// Byte 31 : 
// Byte 32 : 
// Byte 33 : 
// Byte 34 : REAL  - Data.X2
// Byte 35 : 
// Byte 36 : 
// Byte 37 : 
// Byte 38 : REAL  - Data.Y1
// Byte 39 : 
// Byte 40 : 
// Byte 41 : 
// Byte 42 : REAL  - Data.Y2
// Byte 43 : 
// Byte 44 : 
// Byte 45 : 
// Byte 46 : REAL  - Data.Z1
// Byte 47 : 
// Byte 48 : 
// Byte 49 : 
// Byte 50 : REAL  - Data.Z2
// Byte 51 : 
// Byte 52 : 
// Byte 53 : 
// Byte 54 : REAL  - Data.Radius
// Byte 55 : 
// Byte 56 : 
// Byte 57 : 
// Byte 58 : REAL  - Data.JointLowerLimit.J1
// Byte 59 : 
// Byte 60 : 
// Byte 61 : 
// Byte 62 : REAL  - Data.JointLowerLimit.J2
// Byte 63 : 
// Byte 64 : 
// Byte 65 : 
// Byte 66 : REAL  - Data.JointLowerLimit.J3
// Byte 67 : 
// Byte 68 : 
// Byte 69 : 
// Byte 70 : REAL  - Data.JointLowerLimit.J4
// Byte 71 : 
// Byte 72 : 
// Byte 73 : 
// Byte 74 : REAL  - Data.JointLowerLimit.J5
// Byte 75 : 
// Byte 76 : 
// Byte 77 : 
// Byte 78 : REAL  - Data.JointLowerLimit.J6
// Byte 79 : 
// Byte 80 : 
// Byte 81 : 
// Byte 82 : REAL  - Data.JointLowerLimit.E1
// Byte 83 : 
// Byte 84 : 
// Byte 85 : 
// Byte 86 : REAL  - Data.JointUpperLimit.J1
// Byte 87 : 
// Byte 88 : 
// Byte 89 : 
// Byte 90 : REAL  - Data.JointUpperLimit.J2
// Byte 91 : 
// Byte 92 : 
// Byte 93 : 
// Byte 94 : REAL  - Data.JointUpperLimit.J3
// Byte 95 : 
// Byte 96 : 
// Byte 97 : 
// Byte 98 : REAL  - Data.JointUpperLimit.J4
// Byte 99 : 
// Byte 100 : 
// Byte 101 : 
// Byte 102 : REAL - Data.JointUpperLimit.J5
// Byte 103 : 
// Byte 104 : 
// Byte 105 : 
// Byte 106 : REAL - Data.JointUpperLimit.J6
// Byte 107 : 
// Byte 108 : 
// Byte 109 : 
// Byte 110 : REAL - Data.JointUpperLimit.E1
// Byte 111 : 
// Byte 112 : 
// Byte 113 : 
// Byte 114 : REAL - Data.JointLowerLimit.E2
// Byte 115 : 
// Byte 116 : 
// Byte 117 : 
// Byte 118 : REAL - Data.JointLowerLimit.E3
// Byte 119 : 
// Byte 120 : 
// Byte 121 : 
// Byte 122 : REAL - Data.JointLowerLimit.E4
// Byte 123 : 
// Byte 124 : 
// Byte 125 : 
// Byte 126 : REAL - Data.JointLowerLimit.E5
// Byte 127 : 
// Byte 128 : 
// Byte 129 : 
// Byte 130 : REAL - Data.JointLowerLimit.E6
// Byte 131 : 
// Byte 132 : 
// Byte 133 : 
// Byte 134 : REAL - Data.JointUpperLimit.E2
// Byte 135 : 
// Byte 136 : 
// Byte 137 : 
// Byte 138 : REAL - Data.JointUpperLimit.E3
// Byte 139 : 
// Byte 140 : 
// Byte 141 : 
// Byte 142 : REAL - Data.JointUpperLimit.E4
// Byte 143 : 
// Byte 144 : 
// Byte 145 : 
// Byte 146 : REAL - Data.JointUpperLimit.E5
// Byte 147 : 
// Byte 148 : 
// Byte 149 : 
// Byte 150 : REAL - Data.JointUpperLimit.E6
// Byte 151 : 
// Byte 152 : 
// Byte 153 : 
// Byte 154 : BOOL - DataChanged
// --------------------------
                  // set command parameter 
_command.CmdTyp   :=  CmdType.WriteWorkArea;
_command.ExecMode :=  ExecMode;
_command.ParSeq   := _command.ParSeq;
_command.Priority :=  Priority;
                  
_command.WorkAreaData := _parCmd.WorkAreaData;
_command.WorkAreaNo   := _parCmd.WorkAreaNo;


// copy command data to header
_cmdHeader := _command;
// call base implementation to copy header to payload buffer
CreateCommandPayload := SUPER^.CreateCommandPayload(AxesGroup := AxesGroup);


// Check parameter must be added ? 
IF ( CheckAddParameter(CreateCommandPayload.PayloadPtr))
THEN
  // add command.WorkAreaNo
  CreateCommandPayload.AddUint(_command.WorkAreaNo);
  // inc parameter counter
 _parameterCnt := _parameterCnt + 1;  
END_IF


// Check parameter must be added ? 
IF ( CheckAddParameter(CreateCommandPayload.PayloadPtr))
THEN
  // add command.ToolData.Timestamp.IEC_DATE
  CreateCommandPayload.AddUint(_command.WorkAreaData.Timestamp.IEC_DATE);
  // inc parameter counter
 _parameterCnt := _parameterCnt + 1;  
END_IF


// Check parameter must be added ? 
IF ( CheckAddParameter(CreateCommandPayload.PayloadPtr))
THEN
  // add command.ToolData.Timestamp.IEC_TIME
  CreateCommandPayload.AddTime(_command.WorkAreaData.Timestamp.IEC_TIME);
  // inc parameter counter
 _parameterCnt := _parameterCnt + 1;  
END_IF


// Check parameter must be added ? 
IF ( CheckAddParameter(CreateCommandPayload.PayloadPtr))
THEN
  // add command.WorkAreaData.AreaType
  CreateCommandPayload.AddUsint(_command.WorkAreaData.AreaType);
  // inc parameter counter
 _parameterCnt := _parameterCnt + 1;  
END_IF


// Check parameter must be added ? 
IF ( CheckAddParameter(CreateCommandPayload.PayloadPtr))
THEN
  // add command.WorkAreaData.AreaMode
  CreateCommandPayload.AddBool(_command.WorkAreaData.AreaMode);
  // inc parameter counter
 _parameterCnt := _parameterCnt + 1;  
END_IF


// Check parameter must be added ? 
IF ( CheckAddParameter(CreateCommandPayload.PayloadPtr))
THEN
  // add command.WorkAreaData.ReactionMode
  CreateCommandPayload.AddUsint(_command.WorkAreaData.ReactionMode);
  // inc parameter counter
 _parameterCnt := _parameterCnt + 1;  
END_IF


// Check parameter must be added ? 
IF ( CheckAddParameter(CreateCommandPayload.PayloadPtr))
THEN
  // add command.WorkAreaData.ActiveModification
  CreateCommandPayload.AddBool(_command.WorkAreaData.ActiveModification);
  // inc parameter counter
 _parameterCnt := _parameterCnt + 1;  
END_IF


// Check parameter must be added ? 
IF ( CheckAddParameter(CreateCommandPayload.PayloadPtr))
THEN
  // add command.WorkAreaData.DefinitionMode
  CreateCommandPayload.AddUsint(_command.WorkAreaData.DefinitionMode);
  // inc parameter counter
 _parameterCnt := _parameterCnt + 1;  
END_IF


// Check parameter must be added ? 
IF ( CheckAddParameter(CreateCommandPayload.PayloadPtr))
THEN
  // add command.WorkAreaData.FrameNo
  CreateCommandPayload.AddUsint(_command.WorkAreaData.FrameNo);
  // inc parameter counter
 _parameterCnt := _parameterCnt + 1;  
END_IF


// Check parameter must be added ? 
IF ( CheckAddParameter(CreateCommandPayload.PayloadPtr))
THEN
  // add command.WorkAreaData.ZeroPointX
  CreateCommandPayload.AddReal(_command.WorkAreaData.ZeroPointX);
  // inc parameter counter
 _parameterCnt := _parameterCnt + 1;  
END_IF


// Check parameter must be added ? 
IF ( CheckAddParameter(CreateCommandPayload.PayloadPtr))
THEN
  // add command.WorkAreaData.ZeroPointY
  CreateCommandPayload.AddReal(_command.WorkAreaData.ZeroPointY);
  // inc parameter counter
 _parameterCnt := _parameterCnt + 1;  
END_IF


// Check parameter must be added ? 
IF ( CheckAddParameter(CreateCommandPayload.PayloadPtr))
THEN
  // add command.WorkAreaData.ZeroPointZ
  CreateCommandPayload.AddReal(_command.WorkAreaData.ZeroPointZ);
  // inc parameter counter
 _parameterCnt := _parameterCnt + 1;  
END_IF


// Check parameter must be added ? 
IF ( CheckAddParameter(CreateCommandPayload.PayloadPtr))
THEN
  // add command.WorkAreaData.X.LowerLimit
  CreateCommandPayload.AddReal(_command.WorkAreaData.X.LowerLimit);
  // inc parameter counter
 _parameterCnt := _parameterCnt + 1;  
END_IF


// Check parameter must be added ? 
IF ( CheckAddParameter(CreateCommandPayload.PayloadPtr))
THEN
  // add command.WorkAreaData.X.UpperLimit
  CreateCommandPayload.AddReal(_command.WorkAreaData.X.UpperLimit);
  // inc parameter counter
 _parameterCnt := _parameterCnt + 1;  
END_IF


// Check parameter must be added ? 
IF ( CheckAddParameter(CreateCommandPayload.PayloadPtr))
THEN
  // add command.WorkAreaData.Y.LowerLimit
  CreateCommandPayload.AddReal(_command.WorkAreaData.Y.LowerLimit);
  // inc parameter counter
 _parameterCnt := _parameterCnt + 1;  
END_IF


// Check parameter must be added ? 
IF ( CheckAddParameter(CreateCommandPayload.PayloadPtr))
THEN
  // add command.WorkAreaData.Y.UpperLimit
  CreateCommandPayload.AddReal(_command.WorkAreaData.Y.UpperLimit);
  // inc parameter counter
 _parameterCnt := _parameterCnt + 1;  
END_IF


// Check parameter must be added ? 
IF ( CheckAddParameter(CreateCommandPayload.PayloadPtr))
THEN
  // add command.WorkAreaData.Z.LowerLimit
  CreateCommandPayload.AddReal(_command.WorkAreaData.Z.LowerLimit);
  // inc parameter counter
 _parameterCnt := _parameterCnt + 1;  
END_IF


// Check parameter must be added ? 
IF ( CheckAddParameter(CreateCommandPayload.PayloadPtr))
THEN
  // add command.WorkAreaData.Z.UpperLimit
  CreateCommandPayload.AddReal(_command.WorkAreaData.Z.UpperLimit);
  // inc parameter counter
 _parameterCnt := _parameterCnt + 1;  
END_IF


// Check parameter must be added ? 
IF ( CheckAddParameter(CreateCommandPayload.PayloadPtr))
THEN
  // add command.WorkAreaData.Radius
  CreateCommandPayload.AddReal(_command.WorkAreaData.Radius);
  // inc parameter counter
 _parameterCnt := _parameterCnt + 1;  
END_IF


// Check parameter must be added ? 
IF ( CheckAddParameter(CreateCommandPayload.PayloadPtr))
THEN
  // add command.WorkAreaData.J1Limit.LowerLimit
  CreateCommandPayload.AddReal(_command.WorkAreaData.J1Limit.LowerLimit);
  // inc parameter counter
 _parameterCnt := _parameterCnt + 1;  
END_IF


// Check parameter must be added ? 
IF ( CheckAddParameter(CreateCommandPayload.PayloadPtr))
THEN
  // add command.WorkAreaData.J2Limit.LowerLimit
  CreateCommandPayload.AddReal(_command.WorkAreaData.J2Limit.LowerLimit);
  // inc parameter counter
 _parameterCnt := _parameterCnt + 1;  
END_IF


// Check parameter must be added ? 
IF ( CheckAddParameter(CreateCommandPayload.PayloadPtr))
THEN
  // add command.WorkAreaData.J3Limit.LowerLimit
  CreateCommandPayload.AddReal(_command.WorkAreaData.J3Limit.LowerLimit);
  // inc parameter counter
 _parameterCnt := _parameterCnt + 1;  
END_IF


// Check parameter must be added ? 
IF ( CheckAddParameter(CreateCommandPayload.PayloadPtr))
THEN
  // add command.WorkAreaData.J4Limit.LowerLimit
  CreateCommandPayload.AddReal(_command.WorkAreaData.J4Limit.LowerLimit);
  // inc parameter counter
 _parameterCnt := _parameterCnt + 1;  
END_IF


// Check parameter must be added ? 
IF ( CheckAddParameter(CreateCommandPayload.PayloadPtr))
THEN
  // add command.WorkAreaData.J5Limit.LowerLimit
  CreateCommandPayload.AddReal(_command.WorkAreaData.J5Limit.LowerLimit);
  // inc parameter counter
 _parameterCnt := _parameterCnt + 1;  
END_IF


// Check parameter must be added ? 
IF ( CheckAddParameter(CreateCommandPayload.PayloadPtr))
THEN
  // add command.WorkAreaData.J6Limit.LowerLimit
  CreateCommandPayload.AddReal(_command.WorkAreaData.J6Limit.LowerLimit);
  // inc parameter counter
 _parameterCnt := _parameterCnt + 1;  
END_IF


// Check parameter must be added ? 
IF ( CheckAddParameter(CreateCommandPayload.PayloadPtr))
THEN
  // add command.WorkAreaData.E1Limit.LowerLimit
  CreateCommandPayload.AddReal(_command.WorkAreaData.E1Limit.LowerLimit);
  // inc parameter counter
 _parameterCnt := _parameterCnt + 1;  
END_IF


// Check parameter must be added ? 
IF ( CheckAddParameter(CreateCommandPayload.PayloadPtr))
THEN
  // add command.WorkAreaData.J1Limit.UpperLimit
  CreateCommandPayload.AddReal(_command.WorkAreaData.J1Limit.UpperLimit);
  // inc parameter counter
 _parameterCnt := _parameterCnt + 1;  
END_IF


// Check parameter must be added ? 
IF ( CheckAddParameter(CreateCommandPayload.PayloadPtr))
THEN
  // add command.WorkAreaData.J2Limit.UpperLimit
  CreateCommandPayload.AddReal(_command.WorkAreaData.J2Limit.UpperLimit);
  // inc parameter counter
 _parameterCnt := _parameterCnt + 1;  
END_IF


// Check parameter must be added ? 
IF ( CheckAddParameter(CreateCommandPayload.PayloadPtr))
THEN
  // add command.WorkAreaData.J3Limit.UpperLimit
  CreateCommandPayload.AddReal(_command.WorkAreaData.J3Limit.UpperLimit);
  // inc parameter counter
 _parameterCnt := _parameterCnt + 1;  
END_IF


// Check parameter must be added ? 
IF ( CheckAddParameter(CreateCommandPayload.PayloadPtr))
THEN
  // add command.WorkAreaData.J4Limit.UpperLimit
  CreateCommandPayload.AddReal(_command.WorkAreaData.J4Limit.UpperLimit);
  // inc parameter counter
 _parameterCnt := _parameterCnt + 1;  
END_IF


// Check parameter must be added ? 
IF ( CheckAddParameter(CreateCommandPayload.PayloadPtr))
THEN
  // add command.WorkAreaData.J5Limit.UpperLimit
  CreateCommandPayload.AddReal(_command.WorkAreaData.J5Limit.UpperLimit);
  // inc parameter counter
 _parameterCnt := _parameterCnt + 1;  
END_IF


// Check parameter must be added ? 
IF ( CheckAddParameter(CreateCommandPayload.PayloadPtr))
THEN
  // add command.WorkAreaData.J6Limit.UpperLimit
  CreateCommandPayload.AddReal(_command.WorkAreaData.J6Limit.UpperLimit);
  // inc parameter counter
 _parameterCnt := _parameterCnt + 1;  
END_IF


// Check parameter must be added ? 
IF ( CheckAddParameter(CreateCommandPayload.PayloadPtr))
THEN
  // add command.WorkAreaData.E1Limit.UpperLimit
  CreateCommandPayload.AddReal(_command.WorkAreaData.E1Limit.UpperLimit);
  // inc parameter counter
 _parameterCnt := _parameterCnt + 1;  
END_IF


// Check parameter must be added ? 
IF ( CheckAddParameter(CreateCommandPayload.PayloadPtr))
THEN
  // add command.WorkAreaData.E2Limit.LowerLimit
  CreateCommandPayload.AddReal(_command.WorkAreaData.E2Limit.LowerLimit);
  // inc parameter counter
 _parameterCnt := _parameterCnt + 1;  
END_IF


// Check parameter must be added ? 
IF ( CheckAddParameter(CreateCommandPayload.PayloadPtr))
THEN
  // add command.WorkAreaData.E3Limit.LowerLimit
  CreateCommandPayload.AddReal(_command.WorkAreaData.E3Limit.LowerLimit);
  // inc parameter counter
 _parameterCnt := _parameterCnt + 1;  
END_IF


// Check parameter must be added ? 
IF ( CheckAddParameter(CreateCommandPayload.PayloadPtr))
THEN
  // add command.WorkAreaData.E4Limit.LowerLimit
  CreateCommandPayload.AddReal(_command.WorkAreaData.E4Limit.LowerLimit);
  // inc parameter counter
 _parameterCnt := _parameterCnt + 1;  
END_IF


// Check parameter must be added ? 
IF ( CheckAddParameter(CreateCommandPayload.PayloadPtr))
THEN
  // add command.WorkAreaData.E5Limit.LowerLimit
  CreateCommandPayload.AddReal(_command.WorkAreaData.E5Limit.LowerLimit);
  // inc parameter counter
 _parameterCnt := _parameterCnt + 1;  
END_IF


// Check parameter must be added ? 
IF ( CheckAddParameter(CreateCommandPayload.PayloadPtr))
THEN
  // add command.WorkAreaData.E6Limit.LowerLimit
  CreateCommandPayload.AddReal(_command.WorkAreaData.E6Limit.LowerLimit);
  // inc parameter counter
 _parameterCnt := _parameterCnt + 1;  
END_IF


// Check parameter must be added ? 
IF ( CheckAddParameter(CreateCommandPayload.PayloadPtr))
THEN
  // add command.WorkAreaData.E2Limit.UpperLimit
  CreateCommandPayload.AddReal(_command.WorkAreaData.E2Limit.UpperLimit);
  // inc parameter counter
 _parameterCnt := _parameterCnt + 1;  
END_IF


// Check parameter must be added ? 
IF ( CheckAddParameter(CreateCommandPayload.PayloadPtr))
THEN
  // add command.WorkAreaData.E3Limit.UpperLimit
  CreateCommandPayload.AddReal(_command.WorkAreaData.E3Limit.UpperLimit);
  // inc parameter counter
 _parameterCnt := _parameterCnt + 1;  
END_IF


// Check parameter must be added ? 
IF ( CheckAddParameter(CreateCommandPayload.PayloadPtr))
THEN
  // add command.WorkAreaData.E4Limit.UpperLimit
  CreateCommandPayload.AddReal(_command.WorkAreaData.E4Limit.UpperLimit);
  // inc parameter counter
 _parameterCnt := _parameterCnt + 1;  
END_IF


// Check parameter must be added ? 
IF ( CheckAddParameter(CreateCommandPayload.PayloadPtr))
THEN
  // add command.WorkAreaData.E5Limit.UpperLimit
  CreateCommandPayload.AddReal(_command.WorkAreaData.E5Limit.UpperLimit);
  // inc parameter counter
 _parameterCnt := _parameterCnt + 1;  
END_IF


// Check parameter must be added ? 
IF ( CheckAddParameter(CreateCommandPayload.PayloadPtr))
THEN
  // add command.WorkAreaData.E6Limit.UpperLimit
  CreateCommandPayload.AddReal(_command.WorkAreaData.E6Limit.UpperLimit);
  // inc parameter counter
 _parameterCnt := _parameterCnt + 1;  
END_IF


// Check parameter must be added ? 
IF ( CheckAddParameter(CreateCommandPayload.PayloadPtr))
THEN
  // add command.DataChanged
  CreateCommandPayload.AddBool(_command.DataChanged);
  // inc parameter counter
 _parameterCnt := _parameterCnt + 1;  
END_IF

  
// Create logging
CreateCommandPayloadLog(AxesGroup := AxesGroup, ParameterCnt := _parameterCnt);
                
END_METHOD

METHOD INTERNAL CreateCommandPayloadLog
VAR_IN_OUT
  /// Robot assignment of function
  AxesGroup : AxesGroup; 
END_VAR
VAR_INPUT
  /// Parameter count
  ParameterCnt : DINT;
END_VAR
                  // Create log entry for Parameter start
CreateLogMessagePara1 ( Timestamp   := AxesGroup.State.SystemTime,
                        MessageType := MessageType.CMD,
                        Severity    := Severity.DEBUG,
                        MessageCode := 0,
                        MessageText := 'Create command payload with {1} parameter(s) :',
                        Para1       := DINT_TO_STRING(ParameterCnt));
                       

// Return if no parameter is remaining...
IF ( ParameterCnt = 0 ) THEN RETURN; END_IF
// dec remaining parameter(s)                        
ParameterCnt := ParameterCnt - 1;
// Create log entry for WorkAreaNo
CreateLogMessagePara1 ( Timestamp   := AxesGroup.State.SystemTime,
                        MessageType := MessageType.CMD,
                        Severity    := Severity.DEBUG,
                        MessageCode := 0,
                        MessageText := 'Command.WorkAreaNo = {1}',
                        Para1       :=  UINT_TO_STRING(_command.WorkAreaNo));


// Return if no parameter is remaining...
IF ( ParameterCnt = 0 ) THEN RETURN; END_IF
// dec remaining parameter(s)                        
ParameterCnt := ParameterCnt - 1;
// Create log entry for WorkAreaData.Timestamp.IEC_DATE
CreateLogMessagePara1 ( Timestamp   := AxesGroup.State.SystemTime,
                        MessageType := MessageType.CMD,
                        Severity    := Severity.DEBUG,
                        MessageCode := 0,
                        MessageText := 'Command.WorkAreaData.Timestamp.IEC_DATE = {1}',
                        Para1       :=  IEC_DATE_TO_STRING(_command.WorkAreaData.Timestamp.IEC_DATE));


// Return if no parameter is remaining...
IF ( ParameterCnt = 0 ) THEN RETURN; END_IF
// dec remaining parameter(s)                        
ParameterCnt := ParameterCnt - 1;
// Create log entry for WorkAreaData.Timestamp.IEC_DATE
CreateLogMessagePara1 ( Timestamp   := AxesGroup.State.SystemTime,
                        MessageType := MessageType.CMD,
                        Severity    := Severity.DEBUG,
                        MessageCode := 0,
                        MessageText := 'Command.WorkAreaData.Timestamp.IEC_TIME = {1}',
                        Para1       :=  IEC_TIME_TO_STRING(_command.WorkAreaData.Timestamp.IEC_TIME));


// Return if no parameter is remaining...
IF ( ParameterCnt = 0 ) THEN RETURN; END_IF
// dec remaining parameter(s)                        
ParameterCnt := ParameterCnt - 1;
// Create log entry for WorkAreaData.AreaType
CreateLogMessagePara1 ( Timestamp   := AxesGroup.State.SystemTime,
                        MessageType := MessageType.CMD,
                        Severity    := Severity.DEBUG,
                        MessageCode := 0,
                        MessageText := 'Command.WorkAreaData.AreaType = {1}',
                        Para1       :=  AREA_TYPE_TO_STRING(_command.WorkAreaData.AreaType));


// Return if no parameter is remaining...
IF ( ParameterCnt = 0 ) THEN RETURN; END_IF
// dec remaining parameter(s)                        
ParameterCnt := ParameterCnt - 1;
// Create log entry for WorkAreaData.AreaMode
CreateLogMessagePara1 ( Timestamp   := AxesGroup.State.SystemTime,
                        MessageType := MessageType.CMD,
                        Severity    := Severity.DEBUG,
                        MessageCode := 0,
                        MessageText := 'Command.WorkAreaData.AreaMode = {1}',
                        Para1       :=  BOOL_TO_STRING(_command.WorkAreaData.AreaMode));


// Return if no parameter is remaining...
IF ( ParameterCnt = 0 ) THEN RETURN; END_IF
// dec remaining parameter(s)                        
ParameterCnt := ParameterCnt - 1;
// Create log entry for WorkAreaData.ReactionMode
CreateLogMessagePara1 ( Timestamp   := AxesGroup.State.SystemTime,
                        MessageType := MessageType.CMD,
                        Severity    := Severity.DEBUG,
                        MessageCode := 0,
                        MessageText := 'Command.WorkAreaData.ReactionMode = {1}',
                        Para1       := WORK_AREA_REACTION_MODE_TO_STRING(_command.WorkAreaData.ReactionMode));


// Return if no parameter is remaining...
IF ( ParameterCnt = 0 ) THEN RETURN; END_IF
// dec remaining parameter(s)                        
ParameterCnt := ParameterCnt - 1;
// Create log entry for WorkAreaData.ActiveModification
CreateLogMessagePara1 ( Timestamp   := AxesGroup.State.SystemTime,
                        MessageType := MessageType.CMD,
                        Severity    := Severity.DEBUG,
                        MessageCode := 0,
                        MessageText := 'Command.WorkAreaData.ActiveModification = {1}',
                        Para1       := BOOL_TO_STRING(_command.WorkAreaData.ActiveModification));


// Return if no parameter is remaining...
IF ( ParameterCnt = 0 ) THEN RETURN; END_IF
// dec remaining parameter(s)                        
ParameterCnt := ParameterCnt - 1;
// Create log entry for WorkAreaData.DefinitionMode
CreateLogMessagePara1 ( Timestamp   := AxesGroup.State.SystemTime,
                        MessageType := MessageType.CMD,
                        Severity    := Severity.DEBUG,
                        MessageCode := 0,
                        MessageText := 'Command.WorkAreaData.DefinitionMode = {1}',
                        Para1       := DEFINITION_MODE_TO_STRING(_command.WorkAreaData.DefinitionMode));


// Return if no parameter is remaining...
IF ( ParameterCnt = 0 ) THEN RETURN; END_IF
// dec remaining parameter(s)                        
ParameterCnt := ParameterCnt - 1;
// Create log entry for WorkAreaData.FrameNo
CreateLogMessagePara1 ( Timestamp   := AxesGroup.State.SystemTime,
                        MessageType := MessageType.CMD,
                        Severity    := Severity.DEBUG,
                        MessageCode := 0,
                        MessageText := 'Command.WorkAreaData.FrameNo = {1}',
                        Para1       := USINT_TO_STRING(_command.WorkAreaData.FrameNo));


// Return if no parameter is remaining...
IF ( ParameterCnt = 0 ) THEN RETURN; END_IF
// dec remaining parameter(s)                        
ParameterCnt := ParameterCnt - 1;
// Create log entry for WorkAreaData.ZeroPointX
CreateLogMessagePara1 ( Timestamp   := AxesGroup.State.SystemTime,
                        MessageType := MessageType.CMD,
                        Severity    := Severity.DEBUG,
                        MessageCode := 0,
                        MessageText := 'Command.WorkAreaData.ZeroPointX = {1}',
                        Para1       := REAL_TO_STRING(_command.WorkAreaData.ZeroPointX));


// Return if no parameter is remaining...
IF ( ParameterCnt = 0 ) THEN RETURN; END_IF
// dec remaining parameter(s)                        
ParameterCnt := ParameterCnt - 1;
// Create log entry for WorkAreaData.ZeroPointY
CreateLogMessagePara1 ( Timestamp   := AxesGroup.State.SystemTime,
                        MessageType := MessageType.CMD,
                        Severity    := Severity.DEBUG,
                        MessageCode := 0,
                        MessageText := 'Command.WorkAreaData.ZeroPointY = {1}',
                        Para1       := REAL_TO_STRING(_command.WorkAreaData.ZeroPointY));


// Return if no parameter is remaining...
IF ( ParameterCnt = 0 ) THEN RETURN; END_IF
// dec remaining parameter(s)                        
ParameterCnt := ParameterCnt - 1;
// Create log entry for WorkAreaData.ZeroPointZ
CreateLogMessagePara1 ( Timestamp   := AxesGroup.State.SystemTime,
                        MessageType := MessageType.CMD,
                        Severity    := Severity.DEBUG,
                        MessageCode := 0,
                        MessageText := 'Command.WorkAreaData.ZeroPointZ = {1}',
                        Para1       := REAL_TO_STRING(_command.WorkAreaData.ZeroPointZ));


// Return if no parameter is remaining...
IF ( ParameterCnt = 0 ) THEN RETURN; END_IF
// dec remaining parameter(s)                        
ParameterCnt := ParameterCnt - 1;
// Create log entry for WorkAreaData.X.LowerLimit
CreateLogMessagePara1 ( Timestamp   := AxesGroup.State.SystemTime,
                        MessageType := MessageType.CMD,
                        Severity    := Severity.DEBUG,
                        MessageCode := 0,
                        MessageText := 'Command.WorkAreaData.X.LowerLimit = {1}',
                        Para1       := REAL_TO_STRING(_command.WorkAreaData.X.LowerLimit));


// Return if no parameter is remaining...
IF ( ParameterCnt = 0 ) THEN RETURN; END_IF
// dec remaining parameter(s)                        
ParameterCnt := ParameterCnt - 1;
// Create log entry for WorkAreaData.X.UpperLimit
CreateLogMessagePara1 ( Timestamp   := AxesGroup.State.SystemTime,
                        MessageType := MessageType.CMD,
                        Severity    := Severity.DEBUG,
                        MessageCode := 0,
                        MessageText := 'Command.WorkAreaData.X.UpperLimit = {1}',
                        Para1       := REAL_TO_STRING(_command.WorkAreaData.X.UpperLimit));


// Return if no parameter is remaining...
IF ( ParameterCnt = 0 ) THEN RETURN; END_IF
// dec remaining parameter(s)                        
ParameterCnt := ParameterCnt - 1;
// Create log entry for WorkAreaData.Y.LowerLimit
CreateLogMessagePara1 ( Timestamp   := AxesGroup.State.SystemTime,
                        MessageType := MessageType.CMD,
                        Severity    := Severity.DEBUG,
                        MessageCode := 0,
                        MessageText := 'Command.WorkAreaData.Y.LowerLimit = {1}',
                        Para1       := REAL_TO_STRING(_command.WorkAreaData.Y.LowerLimit));


// Return if no parameter is remaining...
IF ( ParameterCnt = 0 ) THEN RETURN; END_IF
// dec remaining parameter(s)                        
ParameterCnt := ParameterCnt - 1;
// Create log entry for WorkAreaData.Y.UpperLimit
CreateLogMessagePara1 ( Timestamp   := AxesGroup.State.SystemTime,
                        MessageType := MessageType.CMD,
                        Severity    := Severity.DEBUG,
                        MessageCode := 0,
                        MessageText := 'Command.WorkAreaData.Y.UpperLimit = {1}',
                        Para1       := REAL_TO_STRING(_command.WorkAreaData.Y.UpperLimit));


// Return if no parameter is remaining...
IF ( ParameterCnt = 0 ) THEN RETURN; END_IF
// dec remaining parameter(s)                        
ParameterCnt := ParameterCnt - 1;
// Create log entry for WorkAreaData.Z.LowerLimit
CreateLogMessagePara1 ( Timestamp   := AxesGroup.State.SystemTime,
                        MessageType := MessageType.CMD,
                        Severity    := Severity.DEBUG,
                        MessageCode := 0,
                        MessageText := 'Command.WorkAreaData.Z.LowerLimit = {1}',
                        Para1       := REAL_TO_STRING(_command.WorkAreaData.Z.LowerLimit));


// Return if no parameter is remaining...
IF ( ParameterCnt = 0 ) THEN RETURN; END_IF
// dec remaining parameter(s)                        
ParameterCnt := ParameterCnt - 1;
// Create log entry for WorkAreaData.Z.UpperLimit
CreateLogMessagePara1 ( Timestamp   := AxesGroup.State.SystemTime,
                        MessageType := MessageType.CMD,
                        Severity    := Severity.DEBUG,
                        MessageCode := 0,
                        MessageText := 'Command.WorkAreaData.Z.UpperLimit = {1}',
                        Para1       := REAL_TO_STRING(_command.WorkAreaData.Z.UpperLimit));


// Return if no parameter is remaining...
IF ( ParameterCnt = 0 ) THEN RETURN; END_IF
// dec remaining parameter(s)                        
ParameterCnt := ParameterCnt - 1;
// Create log entry for WorkAreaData.Radius
CreateLogMessagePara1 ( Timestamp   := AxesGroup.State.SystemTime,
                        MessageType := MessageType.CMD,
                        Severity    := Severity.DEBUG,
                        MessageCode := 0,
                        MessageText := 'Command.WorkAreaData.Radius = {1}',
                        Para1       := REAL_TO_STRING(_command.WorkAreaData.Radius));


// Return if no parameter is remaining...
IF ( ParameterCnt = 0 ) THEN RETURN; END_IF
// dec remaining parameter(s)                        
ParameterCnt := ParameterCnt - 1;
// Create log entry for WorkAreaData.J1Limit.LowerLimit
CreateLogMessagePara1 ( Timestamp   := AxesGroup.State.SystemTime,
                        MessageType := MessageType.CMD,
                        Severity    := Severity.DEBUG,
                        MessageCode := 0,
                        MessageText := 'Command.WorkAreaData.J1Limit.LowerLimit = {1}',
                        Para1       := REAL_TO_STRING(_command.WorkAreaData.J1Limit.LowerLimit));


// Return if no parameter is remaining...
IF ( ParameterCnt = 0 ) THEN RETURN; END_IF
// dec remaining parameter(s)                        
ParameterCnt := ParameterCnt - 1;
// Create log entry for WorkAreaData.J2Limit.LowerLimit
CreateLogMessagePara1 ( Timestamp   := AxesGroup.State.SystemTime,
                        MessageType := MessageType.CMD,
                        Severity    := Severity.DEBUG,
                        MessageCode := 0,
                        MessageText := 'Command.WorkAreaData.J2Limit.LowerLimit = {1}',
                        Para1       := REAL_TO_STRING(_command.WorkAreaData.J2Limit.LowerLimit));


// Return if no parameter is remaining...
IF ( ParameterCnt = 0 ) THEN RETURN; END_IF
// dec remaining parameter(s)                        
ParameterCnt := ParameterCnt - 1;
// Create log entry for WorkAreaData.J3Limit.LowerLimit
CreateLogMessagePara1 ( Timestamp   := AxesGroup.State.SystemTime,
                        MessageType := MessageType.CMD,
                        Severity    := Severity.DEBUG,
                        MessageCode := 0,
                        MessageText := 'Command.WorkAreaData.J3Limit.LowerLimit = {1}',
                        Para1       := REAL_TO_STRING(_command.WorkAreaData.J3Limit.LowerLimit));


